SPLINE
SPL {X  -137.039, Y  +756.986, Z    +0.000, E1   -45.206, E3 +141112.390}
SPL {X  -152.094, Y  +724.074, Z    +0.000, E1   -34.132, E3 +141128.337}
SPL {X  -158.930, Y  +692.872, Z    +0.000, E1   -16.505, E3 +141134.653}
SPL {X  -160.000, Y  +673.072, Z    +0.000, E1    -0.858, E3 +141135.963}
SPL {X  -160.000, Y  +670.505, Z    +0.000, E1    +2.991, E3 +141136.000}
SPL {X  -160.000, Y  +665.157, Z    +0.000, E1   +13.199, E3 +141136.230}
SPL {X  -160.000, Y  +657.552, Z    +0.000, E1   +28.428, E3 +141136.915}
SPL {X  -160.000, Y  +642.088, Z    +0.000, E1   +49.428, E3 +141139.905}
SPL {X  -160.000, Y  +582.331, Z    +0.000, E1   +67.139, E3 +141162.371}
SPL {X  -160.000, Y  +443.344, Z    +0.000, E1   +69.515, E3 +141246.858}
SPL {X  -160.000, Y  +423.295, Z    +0.000, E1   +69.546, E3 +141262.678}
SPL {X  -155.937, Y  +349.874, Z    +0.000, E1   +73.941, E3 +141270.748}
SPL {X  -155.646, Y  +348.628, Z    +0.000, E1   +73.073, E3 +141280.631}
SPL {X  -155.163, Y  +346.655, Z    +0.000, E1   +71.976, E3 +141292.619}
SPL {X  -154.105, Y  +342.669, Z    +0.000, E1   +70.814, E3 +141306.124}
SPL {X  -152.951, Y  +338.733, Z    +0.000, E1   +69.529, E3 +141319.967}
SPL {X  -150.673, Y  +331.871, Z    +0.000, E1   +68.778, E3 +141331.215}
SPL {X  -146.876, Y  +322.238, Z    +0.000, E1   +68.294, E3 +141342.396}
SPL {X  -142.952, Y  +313.834, Z    +0.000, E1   +67.744, E3 +141352.675}
SPL {X  -139.245, Y  +306.891, Z    +0.000, E1   +67.208, E3 +141361.459}
SPL {X  -135.108, Y  +299.992, Z    +0.000, E1   +66.599, E3 +141370.410}
SPL {X  -130.642, Y  +293.328, Z    +0.000, E1   +65.888, E3 +141379.263}
SPL {X  -126.461, Y  +287.682, Z    +0.000, E1   +65.179, E3 +141386.826}
SPL {X   -93.259, Y  +255.690, Z    +0.000, E1   +54.095, E3 +141502.207}
ENDSPLINE

SPLINE
SPL {X  -130.811, Y  +293.568, Z    +0.000, E1   +46.951, E3 +141646.068}
SPL {X  -151.580, Y  +334.479, Z    +0.000, E1   +34.520, E3 +141670.191}
SPL {X  -157.897, Y  +359.846, Z    +0.000, E1   +21.040, E3 +141676.148}
SPL {X  -159.671, Y  +375.443, Z    +0.000, E1   +10.084, E3 +141677.964}
SPL {X  -160.000, Y  +387.403, Z    +0.000, E1    +0.377, E3 +141678.439}
SPL {X  -160.000, Y  +391.807, Z    +0.000, E1    -7.102, E3 +141678.543}
SPL {X  -160.000, Y  +398.244, Z    +0.000, E1   -19.803, E3 +141678.977}
SPL {X  -160.000, Y  +410.795, Z    +0.000, E1   -41.112, E3 +141680.790}
SPL {X  -160.000, Y  +461.796, Z    +0.000, E1   -65.564, E3 +141697.433}
SPL {X  -160.000, Y  +623.854, Z    +0.000, E1   -69.845, E3 +141791.505}
SPL {X  -160.000, Y  +641.581, Z    +0.000, E1   -69.837, E3 +141805.345}
SPL {X  -160.000, Y  +657.932, Z    +0.000, E1   -69.833, E3 +141818.103}
SPL {X  -159.989, Y  +676.310, Z    +0.000, E1   -69.844, E3 +141832.411}
SPL {X  -158.945, Y  +692.747, Z    +0.000, E1   -69.717, E3 +141846.339}
SPL {X  -156.998, Y  +705.248, Z    +0.000, E1   -69.481, E3 +141858.126}
SPL {X  -153.152, Y  +720.707, Z    +0.000, E1   -69.072, E3 +141874.038}
SPL {X  -148.823, Y  +733.152, Z    +0.000, E1   -68.450, E3 +141888.196}
SPL {X  -145.304, Y  +741.384, Z    +0.000, E1   -67.989, E3 +141897.996}
SPL {X  -141.481, Y  +749.119, Z    +0.000, E1   -67.448, E3 +141907.621}
SPL {X  -137.717, Y  +755.849, Z    +0.000, E1   -66.896, E3 +141916.255}
SPL {X  -133.615, Y  +762.417, Z    +0.000, E1   -66.275, E3 +141924.870}
SPL {X  -128.952, Y  +769.117, Z    +0.000, E1   -65.522, E3 +141933.832}
SPL {X  -125.615, Y  +773.501, Z    +0.000, E1   -64.909, E3 +141939.768}
SPL {X   -93.482, Y  +804.250, Z    +0.000, E1   -52.853, E3 +142076.966}
ENDSPLINE

SPLINE
SPL {X  -137.039, Y  +756.986, Z    +0.000, E1   -45.206, E3 +142207.629}
SPL {X  -152.094, Y  +724.074, Z    +0.000, E1   -34.132, E3 +142223.576}
SPL {X  -158.930, Y  +692.872, Z    +0.000, E1   -16.505, E3 +142229.892}
SPL {X  -160.000, Y  +673.072, Z    +0.000, E1    -0.858, E3 +142231.202}
SPL {X  -160.000, Y  +670.505, Z    +0.000, E1    +2.991, E3 +142231.239}
SPL {X  -160.000, Y  +665.157, Z    +0.000, E1   +13.199, E3 +142231.468}
SPL {X  -160.000, Y  +657.552, Z    +0.000, E1   +28.428, E3 +142232.153}
SPL {X  -160.000, Y  +642.088, Z    +0.000, E1   +49.428, E3 +142235.143}
SPL {X  -160.000, Y  +582.331, Z    +0.000, E1   +67.139, E3 +142257.610}
SPL {X  -160.000, Y  +443.344, Z    +0.000, E1   +69.515, E3 +142342.096}
SPL {X  -160.000, Y  +423.295, Z    +0.000, E1   +69.546, E3 +142357.917}
SPL {X  -155.937, Y  +349.874, Z    +0.000, E1   +73.941, E3 +142365.987}
SPL {X  -155.646, Y  +348.628, Z    +0.000, E1   +73.073, E3 +142375.870}
SPL {X  -155.163, Y  +346.655, Z    +0.000, E1   +71.976, E3 +142387.858}
SPL {X  -154.105, Y  +342.669, Z    +0.000, E1   +70.814, E3 +142401.363}
SPL {X  -152.951, Y  +338.733, Z    +0.000, E1   +69.529, E3 +142415.206}
SPL {X  -150.673, Y  +331.871, Z    +0.000, E1   +68.778, E3 +142426.454}
SPL {X  -146.876, Y  +322.238, Z    +0.000, E1   +68.294, E3 +142437.635}
SPL {X  -142.952, Y  +313.834, Z    +0.000, E1   +67.744, E3 +142447.914}
SPL {X  -139.245, Y  +306.891, Z    +0.000, E1   +67.208, E3 +142456.698}
SPL {X  -135.108, Y  +299.992, Z    +0.000, E1   +66.599, E3 +142465.649}
SPL {X  -130.642, Y  +293.328, Z    +0.000, E1   +65.888, E3 +142474.501}
SPL {X  -126.461, Y  +287.682, Z    +0.000, E1   +65.179, E3 +142482.064}
SPL {X   -93.259, Y  +255.690, Z    +0.000, E1   +54.095, E3 +142597.446}
ENDSPLINE

SPLINE
SPL {X  -130.811, Y  +293.568, Z    +0.000, E1   +46.951, E3 +142741.307}
SPL {X  -151.580, Y  +334.479, Z    +0.000, E1   +34.520, E3 +142765.429}
SPL {X  -157.897, Y  +359.846, Z    +0.000, E1   +21.040, E3 +142771.387}
SPL {X  -159.671, Y  +375.443, Z    +0.000, E1   +10.084, E3 +142773.202}
SPL {X  -160.000, Y  +387.403, Z    +0.000, E1    +0.377, E3 +142773.678}
SPL {X  -160.000, Y  +391.807, Z    +0.000, E1    -7.102, E3 +142773.782}
SPL {X  -160.000, Y  +398.244, Z    +0.000, E1   -19.803, E3 +142774.216}
SPL {X  -160.000, Y  +410.795, Z    +0.000, E1   -41.112, E3 +142776.029}
SPL {X  -160.000, Y  +461.796, Z    +0.000, E1   -65.564, E3 +142792.672}
SPL {X  -160.000, Y  +623.854, Z    +0.000, E1   -69.845, E3 +142886.744}
SPL {X  -160.000, Y  +641.581, Z    +0.000, E1   -69.837, E3 +142900.583}
SPL {X  -160.000, Y  +657.932, Z    +0.000, E1   -69.833, E3 +142913.342}
SPL {X  -159.989, Y  +676.310, Z    +0.000, E1   -69.844, E3 +142927.650}
SPL {X  -158.945, Y  +692.747, Z    +0.000, E1   -69.717, E3 +142941.578}
SPL {X  -156.998, Y  +705.248, Z    +0.000, E1   -69.481, E3 +142953.365}
SPL {X  -153.152, Y  +720.707, Z    +0.000, E1   -69.072, E3 +142969.276}
SPL {X  -148.823, Y  +733.152, Z    +0.000, E1   -68.450, E3 +142983.435}
SPL {X  -145.304, Y  +741.384, Z    +0.000, E1   -67.989, E3 +142993.235}
SPL {X  -141.481, Y  +749.119, Z    +0.000, E1   -67.448, E3 +143002.860}
SPL {X  -137.717, Y  +755.849, Z    +0.000, E1   -66.896, E3 +143011.494}
SPL {X  -133.615, Y  +762.417, Z    +0.000, E1   -66.275, E3 +143020.109}
SPL {X  -128.952, Y  +769.117, Z    +0.000, E1   -65.522, E3 +143029.070}
SPL {X  -125.615, Y  +773.501, Z    +0.000, E1   -64.909, E3 +143035.007}
SPL {X   -93.482, Y  +804.250, Z    +0.000, E1   -52.853, E3 +143172.205}
ENDSPLINE

SPLINE
SPL {X  -137.039, Y  +756.986, Z    +0.000, E1   -45.206, E3 +143302.868}
SPL {X  -152.094, Y  +724.074, Z    +0.000, E1   -34.132, E3 +143318.815}
SPL {X  -158.930, Y  +692.872, Z    +0.000, E1   -16.505, E3 +143325.130}
SPL {X  -160.000, Y  +673.072, Z    +0.000, E1    -0.858, E3 +143326.441}
SPL {X  -160.000, Y  +670.505, Z    +0.000, E1    +2.991, E3 +143326.477}
SPL {X  -160.000, Y  +665.157, Z    +0.000, E1   +13.199, E3 +143326.707}
SPL {X  -160.000, Y  +657.552, Z    +0.000, E1   +28.428, E3 +143327.392}
SPL {X  -160.000, Y  +642.088, Z    +0.000, E1   +49.428, E3 +143330.382}
SPL {X  -160.000, Y  +582.331, Z    +0.000, E1   +67.139, E3 +143352.849}
SPL {X  -160.000, Y  +443.344, Z    +0.000, E1   +69.515, E3 +143437.335}
SPL {X  -160.000, Y  +423.295, Z    +0.000, E1   +69.546, E3 +143453.155}
SPL {X  -155.937, Y  +349.874, Z    +0.000, E1   +73.941, E3 +143461.226}
SPL {X  -155.646, Y  +348.628, Z    +0.000, E1   +73.073, E3 +143471.109}
SPL {X  -155.163, Y  +346.655, Z    +0.000, E1   +71.976, E3 +143483.096}
SPL {X  -154.105, Y  +342.669, Z    +0.000, E1   +70.814, E3 +143496.601}
SPL {X  -152.951, Y  +338.733, Z    +0.000, E1   +69.529, E3 +143510.445}
SPL {X  -150.673, Y  +331.871, Z    +0.000, E1   +68.778, E3 +143521.693}
SPL {X  -146.876, Y  +322.238, Z    +0.000, E1   +68.294, E3 +143532.874}
SPL {X  -142.952, Y  +313.834, Z    +0.000, E1   +67.744, E3 +143543.153}
SPL {X  -139.245, Y  +306.891, Z    +0.000, E1   +67.208, E3 +143551.936}
SPL {X  -135.108, Y  +299.992, Z    +0.000, E1   +66.599, E3 +143560.888}
SPL {X  -130.642, Y  +293.328, Z    +0.000, E1   +65.888, E3 +143569.740}
SPL {X  -126.461, Y  +287.682, Z    +0.000, E1   +65.179, E3 +143577.303}
SPL {X   -93.259, Y  +255.690, Z    +0.000, E1   +54.095, E3 +143692.685}
ENDSPLINE

SPLINE
SPL {X  -130.811, Y  +293.568, Z    +0.000, E1   +46.951, E3 +143836.545}
SPL {X  -151.580, Y  +334.479, Z    +0.000, E1   +34.520, E3 +143860.668}
SPL {X  -157.897, Y  +359.846, Z    +0.000, E1   +21.040, E3 +143866.626}
SPL {X  -159.671, Y  +375.443, Z    +0.000, E1   +10.084, E3 +143868.441}
SPL {X  -160.000, Y  +387.403, Z    +0.000, E1    +0.377, E3 +143868.916}
SPL {X  -160.000, Y  +391.807, Z    +0.000, E1    -7.102, E3 +143869.021}
SPL {X  -160.000, Y  +398.244, Z    +0.000, E1   -19.803, E3 +143869.455}
SPL {X  -160.000, Y  +410.795, Z    +0.000, E1   -41.112, E3 +143871.267}
SPL {X  -160.000, Y  +461.796, Z    +0.000, E1   -65.564, E3 +143887.910}
SPL {X  -160.000, Y  +623.854, Z    +0.000, E1   -69.845, E3 +143981.983}
SPL {X  -160.000, Y  +641.581, Z    +0.000, E1   -69.837, E3 +143995.822}
SPL {X  -160.000, Y  +657.932, Z    +0.000, E1   -69.833, E3 +144008.580}
SPL {X  -159.989, Y  +676.310, Z    +0.000, E1   -69.844, E3 +144022.889}
SPL {X  -158.945, Y  +692.747, Z    +0.000, E1   -69.717, E3 +144036.816}
SPL {X  -156.998, Y  +705.248, Z    +0.000, E1   -69.481, E3 +144048.603}
SPL {X  -153.152, Y  +720.707, Z    +0.000, E1   -69.072, E3 +144064.515}
SPL {X  -148.823, Y  +733.152, Z    +0.000, E1   -68.450, E3 +144078.674}
SPL {X  -145.304, Y  +741.384, Z    +0.000, E1   -67.989, E3 +144088.474}
SPL {X  -141.481, Y  +749.119, Z    +0.000, E1   -67.448, E3 +144098.098}
SPL {X  -137.717, Y  +755.849, Z    +0.000, E1   -66.896, E3 +144106.733}
SPL {X  -133.615, Y  +762.417, Z    +0.000, E1   -66.275, E3 +144115.347}
SPL {X  -128.952, Y  +769.117, Z    +0.000, E1   -65.522, E3 +144124.309}
SPL {X  -125.615, Y  +773.501, Z    +0.000, E1   -64.909, E3 +144130.246}
SPL {X   -93.482, Y  +804.250, Z    +0.000, E1   -52.853, E3 +144267.443}
ENDSPLINE

SPLINE
SPL {X  -137.039, Y  +756.986, Z    +0.000, E1   -45.206, E3 +144398.106}
SPL {X  -152.094, Y  +724.074, Z    +0.000, E1   -34.132, E3 +144414.053}
SPL {X  -158.930, Y  +692.872, Z    +0.000, E1   -16.505, E3 +144420.369}
SPL {X  -160.000, Y  +673.072, Z    +0.000, E1    -0.858, E3 +144421.679}
SPL {X  -160.000, Y  +670.505, Z    +0.000, E1    +2.991, E3 +144421.716}
SPL {X  -160.000, Y  +665.157, Z    +0.000, E1   +13.199, E3 +144421.946}
SPL {X  -160.000, Y  +657.552, Z    +0.000, E1   +28.428, E3 +144422.631}
SPL {X  -160.000, Y  +642.088, Z    +0.000, E1   +49.428, E3 +144425.621}
SPL {X  -160.000, Y  +582.331, Z    +0.000, E1   +67.139, E3 +144448.087}
SPL {X  -160.000, Y  +443.344, Z    +0.000, E1   +69.515, E3 +144532.574}
SPL {X  -160.000, Y  +423.295, Z    +0.000, E1   +69.546, E3 +144548.394}
SPL {X  -155.937, Y  +349.874, Z    +0.000, E1   +73.941, E3 +144556.464}
SPL {X  -155.646, Y  +348.628, Z    +0.000, E1   +73.073, E3 +144566.347}
SPL {X  -155.163, Y  +346.655, Z    +0.000, E1   +71.976, E3 +144578.335}
SPL {X  -154.105, Y  +342.669, Z    +0.000, E1   +70.814, E3 +144591.840}
SPL {X  -152.951, Y  +338.733, Z    +0.000, E1   +69.529, E3 +144605.683}
ENDSPLINE

SPLINE
SPL {X  -155.937, Y  +349.872, Z    +0.000, E1   +65.931, E3 +143624.970}
SPL {X  -152.875, Y  +338.486, Z    +0.000, E1   +65.488, E3 +143638.669}
SPL {X  -149.360, Y  +328.327, Z    +0.000, E1   +64.994, E3 +143651.576}
SPL {X  -145.195, Y  +318.481, Z    +0.000, E1   +64.365, E3 +143664.729}
SPL {X  -140.564, Y  +309.268, Z    +0.000, E1   +63.646, E3 +143677.550}
SPL {X  -135.770, Y  +301.044, Z    +0.000, E1   +62.840, E3 +143689.422}
SPL {X  -130.944, Y  +293.756, Z    +0.000, E1   +61.990, E3 +143700.165}
SPL {X  -103.957, Y  +264.074, Z    +0.000, E1   +52.557, E3 +143806.269}
ENDSPLINE

SPLINE
SPL {X  -133.093, Y  +296.896, Z    +0.000, E1   +44.059, E3 +143931.102}
SPL {X  -150.601, Y  +331.670, Z    +0.000, E1   +33.435, E3 +143955.365}
SPL {X  -157.739, Y  +358.898, Z    +0.000, E1   +20.026, E3 +143963.593}
SPL {X  -159.601, Y  +374.403, Z    +0.000, E1   +10.058, E3 +143965.908}
SPL {X  -159.993, Y  +384.251, Z    +0.000, E1    +2.830, E3 +143966.540}
SPL {X  -160.000, Y  +387.929, Z    +0.000, E1    -0.363, E3 +143966.609}
SPL {X  -160.000, Y  +392.137, Z    +0.000, E1    -6.580, E3 +143966.748}
SPL {X  -160.000, Y  +398.334, Z    +0.000, E1   -17.404, E3 +143967.239}
SPL {X  -160.000, Y  +410.558, Z    +0.000, E1   -36.649, E3 +143969.342}
SPL {X  -160.000, Y  +459.534, Z    +0.000, E1   -61.429, E3 +143988.937}
SPL {X  -160.000, Y  +586.246, Z    +0.000, E1   -66.315, E3 +144075.436}
SPL {X  -160.000, Y  +602.823, Z    +0.000, E1   -66.332, E3 +144090.840}
SPL {X  -160.000, Y  +621.796, Z    +0.000, E1   -66.332, E3 +144108.509}
SPL {X  -160.000, Y  +638.226, Z    +0.000, E1   -66.314, E3 +144123.837}
SPL {X  -160.000, Y  +655.092, Z    +0.000, E1   -66.336, E3 +144139.495}
SPL {X  -160.000, Y  +671.716, Z    +0.000, E1   -66.315, E3 +144155.009}
SPL {X  -159.502, Y  +687.017, Z    +0.000, E1   -66.266, E3 +144169.759}
SPL {X  -157.713, Y  +701.353, Z    +0.000, E1   -66.026, E3 +144184.986}
SPL {X  -155.081, Y  +713.767, Z    +0.000, E1   -65.665, E3 +144199.272}
SPL {X  -152.128, Y  +723.968, Z    +0.000, E1   -65.242, E3 +144211.771}
SPL {X  -148.925, Y  +732.892, Z    +0.000, E1   -64.779, E3 +144223.271}
SPL {X  -144.887, Y  +742.280, Z    +0.000, E1   -64.184, E3 +144235.901}
SPL {X  -140.317, Y  +751.285, Z    +0.000, E1   -63.454, E3 +144248.538}
SPL {X  -135.706, Y  +759.158, Z    +0.000, E1   -62.682, E3 +144259.939}
SPL {X  -131.040, Y  +766.207, Z    +0.000, E1   -61.854, E3 +144270.371}
SPL {X  -102.962, Y  +796.870, Z    +0.000, E1   -51.620, E3 +144395.703}
ENDSPLINE

SPLINE
SPL {X  -139.855, Y  +752.122, Z    +0.000, E1   -42.075, E3 +144518.631}
SPL {X  -153.268, Y  +720.324, Z    +0.000, E1   -30.648, E3 +144534.877}
SPL {X  -158.910, Y  +693.048, Z    +0.000, E1   -15.531, E3 +144540.948}
SPL {X  -159.977, Y  +677.095, Z    +0.000, E1    -3.968, E3 +144542.371}
SPL {X  -160.000, Y  +672.556, Z    +0.000, E1    -0.073, E3 +144542.473}
SPL {X  -160.000, Y  +669.399, Z    +0.000, E1    +3.976, E3 +144542.553}
SPL {X  -160.000, Y  +661.045, Z    +0.000, E1   +19.300, E3 +144543.142}
SPL {X  -160.000, Y  +646.999, Z    +0.000, E1   +41.048, E3 +144545.559}
SPL {X  -160.000, Y  +594.464, Z    +0.000, E1   +63.651, E3 +144565.860}
SPL {X  -160.000, Y  +465.200, Z    +0.000, E1   +67.027, E3 +144654.430}
SPL {X  -160.000, Y  +444.745, Z    +0.000, E1   +67.032, E3 +144672.838}
SPL {X  -160.000, Y  +422.224, Z    +0.000, E1   +67.044, E3 +144693.090}
ENDSPLINE

SPLINE
SPL {X  -160.000, Y  +424.635, Z    +0.000, E1   +64.425, E3 +144711.117}
ENDSPLINE

SPLINE
SPL {X  -160.000, Y  +410.501, Z    +0.000, E1   +64.162, E3 +144727.661}
SPL {X  -160.000, Y  +387.965, Z    +0.000, E1   +65.039, E3 +144743.613}
SPL {X  -158.836, Y  +366.435, Z    +0.000, E1   +65.805, E3 +144758.554}
SPL {X  -155.922, Y  +349.806, Z    +0.000, E1   +65.927, E3 +144773.200}
SPL {X  -152.875, Y  +338.486, Z    +0.000, E1   +65.488, E3 +144786.817}
SPL {X  -149.360, Y  +328.327, Z    +0.000, E1   +64.994, E3 +144799.724}
SPL {X  -145.195, Y  +318.481, Z    +0.000, E1   +64.365, E3 +144812.877}
SPL {X  -140.564, Y  +309.268, Z    +0.000, E1   +63.646, E3 +144825.698}
SPL {X  -135.770, Y  +301.044, Z    +0.000, E1   +62.840, E3 +144837.569}
SPL {X  -130.944, Y  +293.756, Z    +0.000, E1   +61.990, E3 +144848.313}
SPL {X  -103.957, Y  +264.074, Z    +0.000, E1   +52.557, E3 +144954.416}
ENDSPLINE

SPLINE
SPL {X  -133.093, Y  +296.896, Z    +0.000, E1   +44.059, E3 +145079.250}
SPL {X  -150.601, Y  +331.670, Z    +0.000, E1   +33.435, E3 +145103.513}
SPL {X  -157.739, Y  +358.898, Z    +0.000, E1   +20.026, E3 +145111.741}
SPL {X  -159.601, Y  +374.403, Z    +0.000, E1   +10.058, E3 +145114.056}
SPL {X  -159.993, Y  +384.251, Z    +0.000, E1    +2.830, E3 +145114.688}
SPL {X  -160.000, Y  +387.929, Z    +0.000, E1    -0.363, E3 +145114.757}
SPL {X  -160.000, Y  +392.137, Z    +0.000, E1    -6.580, E3 +145114.895}
SPL {X  -160.000, Y  +398.334, Z    +0.000, E1   -17.404, E3 +145115.387}
SPL {X  -160.000, Y  +410.558, Z    +0.000, E1   -36.649, E3 +145117.490}
SPL {X  -160.000, Y  +459.534, Z    +0.000, E1   -61.429, E3 +145137.085}
SPL {X  -160.000, Y  +586.246, Z    +0.000, E1   -66.315, E3 +145223.584}
SPL {X  -160.000, Y  +602.823, Z    +0.000, E1   -66.332, E3 +145238.988}
SPL {X  -160.000, Y  +621.796, Z    +0.000, E1   -66.332, E3 +145256.657}
SPL {X  -160.000, Y  +638.226, Z    +0.000, E1   -66.314, E3 +145271.984}
SPL {X  -160.000, Y  +655.092, Z    +0.000, E1   -66.336, E3 +145287.643}
SPL {X  -160.000, Y  +671.716, Z    +0.000, E1   -66.315, E3 +145303.157}
SPL {X  -159.502, Y  +687.017, Z    +0.000, E1   -66.266, E3 +145317.907}
SPL {X  -157.713, Y  +701.353, Z    +0.000, E1   -66.026, E3 +145333.134}
SPL {X  -155.081, Y  +713.767, Z    +0.000, E1   -65.665, E3 +145347.420}
SPL {X  -152.128, Y  +723.968, Z    +0.000, E1   -65.242, E3 +145359.919}
SPL {X  -148.925, Y  +732.892, Z    +0.000, E1   -64.779, E3 +145371.419}
SPL {X  -144.887, Y  +742.280, Z    +0.000, E1   -64.184, E3 +145384.049}
SPL {X  -140.317, Y  +751.285, Z    +0.000, E1   -63.454, E3 +145396.686}
SPL {X  -135.706, Y  +759.158, Z    +0.000, E1   -62.682, E3 +145408.087}
SPL {X  -131.040, Y  +766.207, Z    +0.000, E1   -61.854, E3 +145418.519}
SPL {X  -102.962, Y  +796.870, Z    +0.000, E1   -51.620, E3 +145543.851}
ENDSPLINE

SPLINE
SPL {X  -139.855, Y  +752.122, Z    +0.000, E1   -42.075, E3 +145666.779}
SPL {X  -153.268, Y  +720.324, Z    +0.000, E1   -30.648, E3 +145683.025}
SPL {X  -158.910, Y  +693.048, Z    +0.000, E1   -15.531, E3 +145689.096}
SPL {X  -159.977, Y  +677.095, Z    +0.000, E1    -3.968, E3 +145690.519}
SPL {X  -160.000, Y  +672.556, Z    +0.000, E1    -0.073, E3 +145690.621}
SPL {X  -160.000, Y  +669.399, Z    +0.000, E1    +3.976, E3 +145690.701}
SPL {X  -160.000, Y  +661.045, Z    +0.000, E1   +19.300, E3 +145691.290}
SPL {X  -160.000, Y  +646.999, Z    +0.000, E1   +41.048, E3 +145693.707}
SPL {X  -160.000, Y  +594.464, Z    +0.000, E1   +63.651, E3 +145714.007}
SPL {X  -160.000, Y  +465.200, Z    +0.000, E1   +67.027, E3 +145802.578}
SPL {X  -160.000, Y  +444.745, Z    +0.000, E1   +67.032, E3 +145820.986}
SPL {X  -160.000, Y  +422.224, Z    +0.000, E1   +67.044, E3 +145841.238}
ENDSPLINE

SPLINE
SPL {X  -160.000, Y  +424.635, Z    +0.000, E1   +64.425, E3 +145859.265}
ENDSPLINE

SPLINE
SPL {X  -160.000, Y  +410.501, Z    +0.000, E1   +64.162, E3 +145875.809}
SPL {X  -160.000, Y  +387.965, Z    +0.000, E1   +65.039, E3 +145891.761}
SPL {X  -158.836, Y  +366.435, Z    +0.000, E1   +65.805, E3 +145906.702}
SPL {X  -155.922, Y  +349.806, Z    +0.000, E1   +65.927, E3 +145921.348}
SPL {X  -152.875, Y  +338.486, Z    +0.000, E1   +65.488, E3 +145934.965}
SPL {X  -149.360, Y  +328.327, Z    +0.000, E1   +64.994, E3 +145947.872}
SPL {X  -145.195, Y  +318.481, Z    +0.000, E1   +64.365, E3 +145961.025}
SPL {X  -140.564, Y  +309.268, Z    +0.000, E1   +63.646, E3 +145973.846}
SPL {X  -135.770, Y  +301.044, Z    +0.000, E1   +62.840, E3 +145985.717}
SPL {X  -130.944, Y  +293.756, Z    +0.000, E1   +61.990, E3 +145996.460}
SPL {X  -103.957, Y  +264.074, Z    +0.000, E1   +52.557, E3 +146102.564}
ENDSPLINE

SPLINE
SPL {X  -133.093, Y  +296.896, Z    +0.000, E1   +44.059, E3 +146227.398}
SPL {X  -150.601, Y  +331.670, Z    +0.000, E1   +33.435, E3 +146251.661}
SPL {X  -157.739, Y  +358.898, Z    +0.000, E1   +20.026, E3 +146259.889}
SPL {X  -159.601, Y  +374.403, Z    +0.000, E1   +10.058, E3 +146262.204}
SPL {X  -159.993, Y  +384.251, Z    +0.000, E1    +2.830, E3 +146262.836}
SPL {X  -160.000, Y  +387.929, Z    +0.000, E1    -0.363, E3 +146262.905}
SPL {X  -160.000, Y  +392.137, Z    +0.000, E1    -6.580, E3 +146263.043}
SPL {X  -160.000, Y  +398.334, Z    +0.000, E1   -17.404, E3 +146263.535}
SPL {X  -160.000, Y  +410.558, Z    +0.000, E1   -36.649, E3 +146265.638}
SPL {X  -160.000, Y  +459.534, Z    +0.000, E1   -61.429, E3 +146285.233}
SPL {X  -160.000, Y  +586.246, Z    +0.000, E1   -66.315, E3 +146371.732}
SPL {X  -160.000, Y  +602.823, Z    +0.000, E1   -66.332, E3 +146387.136}
SPL {X  -160.000, Y  +621.796, Z    +0.000, E1   -66.332, E3 +146404.805}
SPL {X  -160.000, Y  +638.226, Z    +0.000, E1   -66.314, E3 +146420.132}
SPL {X  -160.000, Y  +655.092, Z    +0.000, E1   -66.336, E3 +146435.791}
SPL {X  -160.000, Y  +671.716, Z    +0.000, E1   -66.315, E3 +146451.305}
SPL {X  -159.502, Y  +687.017, Z    +0.000, E1   -66.266, E3 +146466.055}
SPL {X  -157.713, Y  +701.353, Z    +0.000, E1   -66.026, E3 +146481.282}
SPL {X  -155.081, Y  +713.767, Z    +0.000, E1   -65.665, E3 +146495.568}
SPL {X  -152.128, Y  +723.968, Z    +0.000, E1   -65.242, E3 +146508.067}
SPL {X  -148.925, Y  +732.892, Z    +0.000, E1   -64.779, E3 +146519.567}
SPL {X  -144.887, Y  +742.280, Z    +0.000, E1   -64.184, E3 +146532.197}
SPL {X  -140.317, Y  +751.285, Z    +0.000, E1   -63.454, E3 +146544.834}
SPL {X  -135.706, Y  +759.158, Z    +0.000, E1   -62.682, E3 +146556.235}
SPL {X  -131.040, Y  +766.207, Z    +0.000, E1   -61.854, E3 +146566.667}
SPL {X  -102.962, Y  +796.870, Z    +0.000, E1   -51.620, E3 +146691.999}
ENDSPLINE

SPLINE
SPL {X  -139.855, Y  +752.122, Z    +0.000, E1   -42.075, E3 +146814.927}
SPL {X  -153.268, Y  +720.324, Z    +0.000, E1   -30.648, E3 +146831.173}
SPL {X  -158.910, Y  +693.048, Z    +0.000, E1   -15.531, E3 +146837.243}
SPL {X  -159.977, Y  +677.095, Z    +0.000, E1    -3.968, E3 +146838.667}
SPL {X  -160.000, Y  +672.556, Z    +0.000, E1    -0.073, E3 +146838.769}
SPL {X  -160.000, Y  +669.399, Z    +0.000, E1    +3.976, E3 +146838.849}
SPL {X  -160.000, Y  +661.045, Z    +0.000, E1   +19.300, E3 +146839.438}
SPL {X  -160.000, Y  +646.999, Z    +0.000, E1   +41.048, E3 +146841.855}
SPL {X  -160.000, Y  +594.464, Z    +0.000, E1   +63.651, E3 +146862.155}
SPL {X  -160.000, Y  +465.200, Z    +0.000, E1   +67.027, E3 +146950.726}
SPL {X  -160.000, Y  +444.745, Z    +0.000, E1   +67.032, E3 +146969.134}
SPL {X  -160.000, Y  +422.224, Z    +0.000, E1   +67.044, E3 +146989.386}
ENDSPLINE

SPLINE
SPL {X  -160.000, Y  +424.635, Z    +0.000, E1   +64.425, E3 +147007.413}
ENDSPLINE

SPLINE
SPL {X  -160.000, Y  +410.501, Z    +0.000, E1   +64.162, E3 +147023.957}
SPL {X  -160.000, Y  +387.965, Z    +0.000, E1   +65.039, E3 +147039.909}
SPL {X  -158.836, Y  +366.435, Z    +0.000, E1   +65.805, E3 +147054.850}
SPL {X  -155.922, Y  +349.806, Z    +0.000, E1   +65.927, E3 +147069.496}
SPL {X  -152.875, Y  +338.486, Z    +0.000, E1   +65.488, E3 +147083.113}
SPL {X  -149.360, Y  +328.327, Z    +0.000, E1   +64.994, E3 +147096.019}
SPL {X  -145.195, Y  +318.481, Z    +0.000, E1   +64.365, E3 +147109.173}
SPL {X  -140.564, Y  +309.268, Z    +0.000, E1   +63.646, E3 +147121.994}
SPL {X  -135.770, Y  +301.044, Z    +0.000, E1   +62.840, E3 +147133.865}
SPL {X  -130.944, Y  +293.756, Z    +0.000, E1   +61.990, E3 +147144.608}
SPL {X  -103.957, Y  +264.074, Z    +0.000, E1   +52.557, E3 +147250.712}
ENDSPLINE

SPLINE
SPL {X  -133.093, Y  +296.896, Z    +0.000, E1   +44.059, E3 +147375.546}
SPL {X  -150.601, Y  +331.670, Z    +0.000, E1   +33.435, E3 +147399.809}
SPL {X  -157.739, Y  +358.898, Z    +0.000, E1   +20.026, E3 +147408.037}
SPL {X  -159.601, Y  +374.403, Z    +0.000, E1   +10.058, E3 +147410.352}
SPL {X  -159.993, Y  +384.251, Z    +0.000, E1    +2.830, E3 +147410.984}
SPL {X  -160.000, Y  +387.929, Z    +0.000, E1    -0.363, E3 +147411.053}
SPL {X  -160.000, Y  +392.137, Z    +0.000, E1    -6.580, E3 +147411.191}
SPL {X  -160.000, Y  +398.334, Z    +0.000, E1   -17.404, E3 +147411.683}
SPL {X  -160.000, Y  +410.558, Z    +0.000, E1   -36.649, E3 +147413.786}
SPL {X  -160.000, Y  +459.534, Z    +0.000, E1   -61.429, E3 +147433.381}
SPL {X  -160.000, Y  +586.246, Z    +0.000, E1   -66.315, E3 +147519.880}
SPL {X  -160.000, Y  +602.823, Z    +0.000, E1   -66.332, E3 +147535.284}
SPL {X  -160.000, Y  +621.796, Z    +0.000, E1   -66.332, E3 +147552.953}
SPL {X  -160.000, Y  +638.226, Z    +0.000, E1   -66.314, E3 +147568.280}
SPL {X  -160.000, Y  +655.092, Z    +0.000, E1   -66.336, E3 +147583.939}
SPL {X  -160.000, Y  +671.716, Z    +0.000, E1   -66.315, E3 +147599.453}
SPL {X  -159.502, Y  +687.017, Z    +0.000, E1   -66.266, E3 +147614.203}
SPL {X  -157.713, Y  +701.353, Z    +0.000, E1   -66.026, E3 +147629.430}
SPL {X  -155.081, Y  +713.767, Z    +0.000, E1   -65.665, E3 +147643.715}
SPL {X  -152.128, Y  +723.968, Z    +0.000, E1   -65.242, E3 +147656.215}
SPL {X  -148.925, Y  +732.892, Z    +0.000, E1   -64.779, E3 +147667.715}
SPL {X  -144.887, Y  +742.280, Z    +0.000, E1   -64.184, E3 +147680.345}
SPL {X  -140.317, Y  +751.285, Z    +0.000, E1   -63.454, E3 +147692.982}
SPL {X  -135.706, Y  +759.158, Z    +0.000, E1   -62.682, E3 +147704.383}
SPL {X  -131.040, Y  +766.207, Z    +0.000, E1   -61.854, E3 +147714.815}
SPL {X  -102.962, Y  +796.870, Z    +0.000, E1   -51.620, E3 +147840.147}
ENDSPLINE

SPLINE
SPL {X  -139.855, Y  +752.122, Z    +0.000, E1   -42.075, E3 +147963.075}
SPL {X  -153.268, Y  +720.324, Z    +0.000, E1   -30.648, E3 +147979.321}
SPL {X  -158.910, Y  +693.048, Z    +0.000, E1   -15.531, E3 +147985.391}
SPL {X  -159.977, Y  +677.095, Z    +0.000, E1    -3.968, E3 +147986.815}
SPL {X  -160.000, Y  +672.556, Z    +0.000, E1    -0.073, E3 +147986.917}
SPL {X  -160.000, Y  +669.399, Z    +0.000, E1    +3.976, E3 +147986.997}
SPL {X  -160.000, Y  +661.045, Z    +0.000, E1   +19.300, E3 +147987.586}
SPL {X  -160.000, Y  +646.999, Z    +0.000, E1   +41.048, E3 +147990.003}
SPL {X  -160.000, Y  +594.464, Z    +0.000, E1   +63.651, E3 +148010.303}
SPL {X  -160.000, Y  +465.200, Z    +0.000, E1   +67.027, E3 +148098.873}
SPL {X  -160.000, Y  +444.745, Z    +0.000, E1   +67.032, E3 +148117.282}
SPL {X  -160.000, Y  +422.224, Z    +0.000, E1   +67.044, E3 +148137.534}
ENDSPLINE

SPLINE
SPL {X  -160.000, Y  +424.635, Z    +0.000, E1   +64.425, E3 +148155.560}
ENDSPLINE

SPLINE
SPL {X  -160.000, Y  +410.501, Z    +0.000, E1   +64.162, E3 +148172.105}
SPL {X  -160.000, Y  +387.965, Z    +0.000, E1   +65.039, E3 +148188.057}
SPL {X  -158.836, Y  +366.435, Z    +0.000, E1   +65.805, E3 +148202.998}
SPL {X  -155.922, Y  +349.806, Z    +0.000, E1   +65.927, E3 +148217.644}
SPL {X  -152.875, Y  +338.486, Z    +0.000, E1   +65.488, E3 +148231.261}
SPL {X  -149.360, Y  +328.327, Z    +0.000, E1   +64.994, E3 +148244.167}
SPL {X  -145.195, Y  +318.481, Z    +0.000, E1   +64.365, E3 +148257.321}
SPL {X  -140.564, Y  +309.268, Z    +0.000, E1   +63.646, E3 +148270.142}
SPL {X  -135.770, Y  +301.044, Z    +0.000, E1   +62.840, E3 +148282.013}
SPL {X  -130.944, Y  +293.756, Z    +0.000, E1   +61.990, E3 +148292.756}
SPL {X  -103.957, Y  +264.074, Z    +0.000, E1   +52.557, E3 +148398.860}
ENDSPLINE

SPLINE
SPL {X  -133.093, Y  +296.896, Z    +0.000, E1   +44.059, E3 +148523.694}
SPL {X  -150.601, Y  +331.670, Z    +0.000, E1   +33.435, E3 +148547.957}
SPL {X  -157.739, Y  +358.898, Z    +0.000, E1   +20.026, E3 +148556.184}
SPL {X  -159.601, Y  +374.403, Z    +0.000, E1   +10.058, E3 +148558.500}
SPL {X  -159.993, Y  +384.251, Z    +0.000, E1    +2.830, E3 +148559.132}
SPL {X  -160.000, Y  +387.929, Z    +0.000, E1    -0.363, E3 +148559.200}
SPL {X  -160.000, Y  +392.137, Z    +0.000, E1    -6.580, E3 +148559.339}
SPL {X  -160.000, Y  +398.334, Z    +0.000, E1   -17.404, E3 +148559.831}
SPL {X  -160.000, Y  +410.558, Z    +0.000, E1   -36.649, E3 +148561.934}
SPL {X  -160.000, Y  +459.534, Z    +0.000, E1   -61.429, E3 +148581.528}
SPL {X  -160.000, Y  +586.246, Z    +0.000, E1   -66.315, E3 +148668.028}
SPL {X  -160.000, Y  +602.823, Z    +0.000, E1   -66.332, E3 +148683.432}
SPL {X  -160.000, Y  +621.796, Z    +0.000, E1   -66.332, E3 +148701.101}
SPL {X  -160.000, Y  +638.226, Z    +0.000, E1   -66.314, E3 +148716.428}
SPL {X  -160.000, Y  +655.092, Z    +0.000, E1   -66.336, E3 +148732.087}
SPL {X  -160.000, Y  +671.716, Z    +0.000, E1   -66.315, E3 +148747.601}
SPL {X  -159.502, Y  +687.017, Z    +0.000, E1   -66.266, E3 +148762.351}
SPL {X  -157.713, Y  +701.353, Z    +0.000, E1   -66.026, E3 +148777.578}
SPL {X  -155.081, Y  +713.767, Z    +0.000, E1   -65.665, E3 +148791.863}
SPL {X  -152.128, Y  +723.968, Z    +0.000, E1   -65.242, E3 +148804.363}
SPL {X  -148.925, Y  +732.892, Z    +0.000, E1   -64.779, E3 +148815.863}
SPL {X  -144.887, Y  +742.280, Z    +0.000, E1   -64.184, E3 +148828.492}
SPL {X  -140.317, Y  +751.285, Z    +0.000, E1   -63.454, E3 +148841.130}
SPL {X  -135.706, Y  +759.158, Z    +0.000, E1   -62.682, E3 +148852.531}
SPL {X  -131.040, Y  +766.207, Z    +0.000, E1   -61.854, E3 +148862.963}
SPL {X  -102.962, Y  +796.870, Z    +0.000, E1   -51.620, E3 +148988.295}
ENDSPLINE

SPLINE
SPL {X  -139.855, Y  +752.122, Z    +0.000, E1   -42.075, E3 +149111.223}
SPL {X  -153.268, Y  +720.324, Z    +0.000, E1   -30.648, E3 +149127.469}
SPL {X  -158.910, Y  +693.048, Z    +0.000, E1   -15.531, E3 +149133.539}
SPL {X  -159.977, Y  +677.095, Z    +0.000, E1    -3.968, E3 +149134.963}
SPL {X  -160.000, Y  +672.556, Z    +0.000, E1    -0.073, E3 +149135.065}
SPL {X  -160.000, Y  +669.399, Z    +0.000, E1    +3.976, E3 +149135.145}
SPL {X  -160.000, Y  +661.045, Z    +0.000, E1   +19.300, E3 +149135.733}
SPL {X  -160.000, Y  +646.999, Z    +0.000, E1   +41.048, E3 +149138.151}
SPL {X  -160.000, Y  +594.464, Z    +0.000, E1   +63.651, E3 +149158.451}
SPL {X  -160.000, Y  +465.200, Z    +0.000, E1   +67.027, E3 +149247.021}
SPL {X  -160.000, Y  +444.745, Z    +0.000, E1   +67.032, E3 +149265.430}
SPL {X  -160.000, Y  +422.224, Z    +0.000, E1   +67.044, E3 +149285.682}
ENDSPLINE

SPLINE
SPL {X  -160.000, Y  +424.635, Z    +0.000, E1   +64.425, E3 +149303.708}
ENDSPLINE

SPLINE
SPL {X  -160.000, Y  +410.501, Z    +0.000, E1   +64.162, E3 +149320.253}
SPL {X  -160.000, Y  +387.965, Z    +0.000, E1   +65.039, E3 +149336.205}
SPL {X  -158.836, Y  +366.435, Z    +0.000, E1   +65.805, E3 +149351.146}
SPL {X  -155.922, Y  +349.806, Z    +0.000, E1   +65.927, E3 +149365.792}
SPL {X  -152.875, Y  +338.486, Z    +0.000, E1   +65.488, E3 +149379.409}
SPL {X  -149.360, Y  +328.327, Z    +0.000, E1   +64.994, E3 +149392.315}
SPL {X  -145.195, Y  +318.481, Z    +0.000, E1   +64.365, E3 +149405.469}
SPL {X  -140.564, Y  +309.268, Z    +0.000, E1   +63.646, E3 +149418.290}
SPL {X  -135.770, Y  +301.044, Z    +0.000, E1   +62.840, E3 +149430.161}
SPL {X  -130.944, Y  +293.756, Z    +0.000, E1   +61.990, E3 +149440.904}
SPL {X  -103.957, Y  +264.074, Z    +0.000, E1   +52.557, E3 +149547.008}
ENDSPLINE

SPLINE
SPL {X  -133.093, Y  +296.896, Z    +0.000, E1   +44.059, E3 +149671.842}
SPL {X  -150.601, Y  +331.670, Z    +0.000, E1   +33.435, E3 +149696.105}
SPL {X  -157.739, Y  +358.898, Z    +0.000, E1   +20.026, E3 +149704.332}
SPL {X  -159.601, Y  +374.403, Z    +0.000, E1   +10.058, E3 +149706.648}
SPL {X  -159.993, Y  +384.251, Z    +0.000, E1    +2.830, E3 +149707.280}
SPL {X  -160.000, Y  +387.929, Z    +0.000, E1    -0.363, E3 +149707.348}
SPL {X  -160.000, Y  +392.137, Z    +0.000, E1    -6.580, E3 +149707.487}
SPL {X  -160.000, Y  +398.334, Z    +0.000, E1   -17.404, E3 +149707.979}
SPL {X  -160.000, Y  +410.558, Z    +0.000, E1   -36.649, E3 +149710.082}
SPL {X  -160.000, Y  +459.534, Z    +0.000, E1   -61.429, E3 +149729.676}
SPL {X  -160.000, Y  +586.246, Z    +0.000, E1   -66.315, E3 +149816.176}
SPL {X  -160.000, Y  +602.823, Z    +0.000, E1   -66.332, E3 +149831.580}
SPL {X  -160.000, Y  +621.796, Z    +0.000, E1   -66.332, E3 +149849.249}
SPL {X  -160.000, Y  +638.226, Z    +0.000, E1   -66.314, E3 +149864.576}
SPL {X  -160.000, Y  +655.092, Z    +0.000, E1   -66.336, E3 +149880.235}
SPL {X  -160.000, Y  +671.716, Z    +0.000, E1   -66.315, E3 +149895.749}
SPL {X  -159.502, Y  +687.017, Z    +0.000, E1   -66.266, E3 +149910.499}
SPL {X  -157.713, Y  +701.353, Z    +0.000, E1   -66.026, E3 +149925.726}
SPL {X  -155.081, Y  +713.767, Z    +0.000, E1   -65.665, E3 +149940.011}
SPL {X  -152.128, Y  +723.968, Z    +0.000, E1   -65.242, E3 +149952.511}
SPL {X  -148.925, Y  +732.892, Z    +0.000, E1   -64.779, E3 +149964.011}
SPL {X  -144.887, Y  +742.280, Z    +0.000, E1   -64.184, E3 +149976.640}
SPL {X  -140.317, Y  +751.285, Z    +0.000, E1   -63.454, E3 +149989.278}
SPL {X  -135.706, Y  +759.158, Z    +0.000, E1   -62.682, E3 +150000.679}
SPL {X  -131.040, Y  +766.207, Z    +0.000, E1   -61.854, E3 +150011.111}
SPL {X  -102.962, Y  +796.870, Z    +0.000, E1   -51.620, E3 +150136.443}
ENDSPLINE

SPLINE
SPL {X  -139.855, Y  +752.122, Z    +0.000, E1   -42.075, E3 +150259.371}
SPL {X  -153.268, Y  +720.324, Z    +0.000, E1   -30.648, E3 +150275.617}
SPL {X  -158.910, Y  +693.048, Z    +0.000, E1   -15.531, E3 +150281.687}
SPL {X  -159.977, Y  +677.095, Z    +0.000, E1    -3.968, E3 +150283.111}
SPL {X  -160.000, Y  +672.556, Z    +0.000, E1    -0.073, E3 +150283.213}
SPL {X  -160.000, Y  +669.399, Z    +0.000, E1    +3.976, E3 +150283.293}
SPL {X  -160.000, Y  +661.045, Z    +0.000, E1   +19.300, E3 +150283.881}
SPL {X  -160.000, Y  +646.999, Z    +0.000, E1   +41.048, E3 +150286.299}
SPL {X  -160.000, Y  +594.464, Z    +0.000, E1   +63.651, E3 +150306.599}
SPL {X  -160.000, Y  +465.200, Z    +0.000, E1   +67.027, E3 +150395.169}
SPL {X  -160.000, Y  +444.745, Z    +0.000, E1   +67.032, E3 +150413.578}
SPL {X  -160.000, Y  +422.224, Z    +0.000, E1   +67.044, E3 +150433.830}
ENDSPLINE

SPLINE
SPL {X  -160.000, Y  +424.635, Z    +0.000, E1   +64.425, E3 +150451.856}
ENDSPLINE

SPLINE
SPL {X  -160.000, Y  +410.501, Z    +0.000, E1   +64.162, E3 +150468.401}
SPL {X  -160.000, Y  +387.965, Z    +0.000, E1   +65.039, E3 +150484.352}
SPL {X  -158.836, Y  +366.435, Z    +0.000, E1   +65.805, E3 +150499.294}
SPL {X  -155.922, Y  +349.806, Z    +0.000, E1   +65.927, E3 +150513.940}
SPL {X  -152.875, Y  +338.486, Z    +0.000, E1   +65.488, E3 +150527.557}
SPL {X  -149.360, Y  +328.327, Z    +0.000, E1   +64.994, E3 +150540.463}
SPL {X  -145.195, Y  +318.481, Z    +0.000, E1   +64.365, E3 +150553.617}
SPL {X  -140.564, Y  +309.268, Z    +0.000, E1   +63.646, E3 +150566.438}
SPL {X  -135.770, Y  +301.044, Z    +0.000, E1   +62.840, E3 +150578.309}
SPL {X  -130.944, Y  +293.756, Z    +0.000, E1   +61.990, E3 +150589.052}
SPL {X  -103.957, Y  +264.074, Z    +0.000, E1   +52.557, E3 +150695.156}
ENDSPLINE

SPLINE
SPL {X  -133.093, Y  +296.896, Z    +0.000, E1   +44.059, E3 +150819.990}
SPL {X  -150.601, Y  +331.670, Z    +0.000, E1   +33.435, E3 +150844.252}
SPL {X  -157.739, Y  +358.898, Z    +0.000, E1   +20.026, E3 +150852.480}
SPL {X  -159.601, Y  +374.403, Z    +0.000, E1   +10.058, E3 +150854.796}
SPL {X  -159.993, Y  +384.251, Z    +0.000, E1    +2.830, E3 +150855.428}
SPL {X  -160.000, Y  +387.929, Z    +0.000, E1    -0.363, E3 +150855.496}
SPL {X  -160.000, Y  +392.137, Z    +0.000, E1    -6.580, E3 +150855.635}
SPL {X  -160.000, Y  +398.334, Z    +0.000, E1   -17.404, E3 +150856.127}
SPL {X  -160.000, Y  +410.558, Z    +0.000, E1   -36.649, E3 +150858.230}
SPL {X  -160.000, Y  +459.534, Z    +0.000, E1   -61.429, E3 +150877.824}
SPL {X  -160.000, Y  +586.246, Z    +0.000, E1   -66.315, E3 +150964.324}
SPL {X  -160.000, Y  +602.823, Z    +0.000, E1   -66.332, E3 +150979.728}
SPL {X  -160.000, Y  +621.796, Z    +0.000, E1   -66.332, E3 +150997.396}
SPL {X  -160.000, Y  +638.226, Z    +0.000, E1   -66.314, E3 +151012.724}
SPL {X  -160.000, Y  +655.092, Z    +0.000, E1   -66.336, E3 +151028.383}
SPL {X  -160.000, Y  +671.716, Z    +0.000, E1   -66.315, E3 +151043.897}
SPL {X  -159.502, Y  +687.017, Z    +0.000, E1   -66.266, E3 +151058.647}
SPL {X  -157.713, Y  +701.353, Z    +0.000, E1   -66.026, E3 +151073.874}
SPL {X  -155.081, Y  +713.767, Z    +0.000, E1   -65.665, E3 +151088.159}
SPL {X  -152.128, Y  +723.968, Z    +0.000, E1   -65.242, E3 +151100.659}
SPL {X  -148.925, Y  +732.892, Z    +0.000, E1   -64.779, E3 +151112.159}
SPL {X  -144.887, Y  +742.280, Z    +0.000, E1   -64.184, E3 +151124.788}
SPL {X  -140.317, Y  +751.285, Z    +0.000, E1   -63.454, E3 +151137.426}
SPL {X  -135.706, Y  +759.158, Z    +0.000, E1   -62.682, E3 +151148.827}
SPL {X  -131.040, Y  +766.207, Z    +0.000, E1   -61.854, E3 +151159.259}
SPL {X  -102.962, Y  +796.870, Z    +0.000, E1   -51.620, E3 +151284.591}
ENDSPLINE

SPLINE
SPL {X  -139.855, Y  +752.122, Z    +0.000, E1   -42.075, E3 +151407.519}
SPL {X  -153.268, Y  +720.324, Z    +0.000, E1   -30.648, E3 +151423.764}
SPL {X  -158.910, Y  +693.048, Z    +0.000, E1   -15.531, E3 +151429.835}
SPL {X  -159.977, Y  +677.095, Z    +0.000, E1    -3.968, E3 +151431.259}
SPL {X  -160.000, Y  +672.556, Z    +0.000, E1    -0.073, E3 +151431.361}
SPL {X  -160.000, Y  +669.399, Z    +0.000, E1    +3.976, E3 +151431.440}
SPL {X  -160.000, Y  +661.045, Z    +0.000, E1   +19.300, E3 +151432.029}
SPL {X  -160.000, Y  +646.999, Z    +0.000, E1   +41.048, E3 +151434.447}
SPL {X  -160.000, Y  +594.464, Z    +0.000, E1   +63.651, E3 +151454.747}
SPL {X  -160.000, Y  +465.200, Z    +0.000, E1   +67.027, E3 +151543.317}
SPL {X  -160.000, Y  +444.745, Z    +0.000, E1   +67.032, E3 +151561.726}
SPL {X  -160.000, Y  +422.224, Z    +0.000, E1   +67.044, E3 +151581.978}
ENDSPLINE

SPLINE
SPL {X  -160.000, Y  +424.635, Z    +0.000, E1   +64.425, E3 +151600.004}
ENDSPLINE

SPLINE
SPL {X  -160.000, Y  +410.501, Z    +0.000, E1   +64.162, E3 +151616.549}
SPL {X  -160.000, Y  +387.965, Z    +0.000, E1   +65.039, E3 +151632.500}
SPL {X  -158.836, Y  +366.435, Z    +0.000, E1   +65.805, E3 +151647.441}
SPL {X  -155.922, Y  +349.806, Z    +0.000, E1   +65.927, E3 +151662.088}
SPL {X  -152.875, Y  +338.486, Z    +0.000, E1   +65.488, E3 +151675.705}
SPL {X  -149.360, Y  +328.327, Z    +0.000, E1   +64.994, E3 +151688.611}
SPL {X  -145.195, Y  +318.481, Z    +0.000, E1   +64.365, E3 +151701.765}
SPL {X  -140.564, Y  +309.268, Z    +0.000, E1   +63.646, E3 +151714.586}
SPL {X  -135.770, Y  +301.044, Z    +0.000, E1   +62.840, E3 +151726.457}
SPL {X  -130.944, Y  +293.756, Z    +0.000, E1   +61.990, E3 +151737.200}
SPL {X  -103.957, Y  +264.074, Z    +0.000, E1   +52.557, E3 +151843.304}
ENDSPLINE

SPLINE
SPL {X  -133.093, Y  +296.896, Z    +0.000, E1   +44.059, E3 +151968.138}
SPL {X  -150.601, Y  +331.670, Z    +0.000, E1   +33.435, E3 +151992.400}
SPL {X  -157.739, Y  +358.898, Z    +0.000, E1   +20.026, E3 +152000.628}
SPL {X  -159.601, Y  +374.403, Z    +0.000, E1   +10.058, E3 +152002.944}
SPL {X  -159.993, Y  +384.251, Z    +0.000, E1    +2.830, E3 +152003.576}
SPL {X  -160.000, Y  +387.929, Z    +0.000, E1    -0.363, E3 +152003.644}
SPL {X  -160.000, Y  +392.137, Z    +0.000, E1    -6.580, E3 +152003.783}
SPL {X  -160.000, Y  +398.334, Z    +0.000, E1   -17.404, E3 +152004.275}
SPL {X  -160.000, Y  +410.558, Z    +0.000, E1   -36.649, E3 +152006.378}
SPL {X  -160.000, Y  +459.534, Z    +0.000, E1   -61.429, E3 +152025.972}
SPL {X  -160.000, Y  +586.246, Z    +0.000, E1   -66.315, E3 +152112.472}
SPL {X  -160.000, Y  +602.823, Z    +0.000, E1   -66.332, E3 +152127.876}
SPL {X  -160.000, Y  +621.796, Z    +0.000, E1   -66.332, E3 +152145.544}
SPL {X  -160.000, Y  +638.226, Z    +0.000, E1   -66.314, E3 +152160.872}
SPL {X  -160.000, Y  +655.092, Z    +0.000, E1   -66.336, E3 +152176.531}
SPL {X  -160.000, Y  +671.716, Z    +0.000, E1   -66.315, E3 +152192.045}
SPL {X  -159.502, Y  +687.017, Z    +0.000, E1   -66.266, E3 +152206.795}
SPL {X  -157.713, Y  +701.353, Z    +0.000, E1   -66.026, E3 +152222.022}
SPL {X  -155.081, Y  +713.767, Z    +0.000, E1   -65.665, E3 +152236.307}
SPL {X  -152.128, Y  +723.968, Z    +0.000, E1   -65.242, E3 +152248.807}
SPL {X  -148.925, Y  +732.892, Z    +0.000, E1   -64.779, E3 +152260.307}
SPL {X  -144.887, Y  +742.280, Z    +0.000, E1   -64.184, E3 +152272.936}
SPL {X  -140.317, Y  +751.285, Z    +0.000, E1   -63.454, E3 +152285.574}
SPL {X  -135.706, Y  +759.158, Z    +0.000, E1   -62.682, E3 +152296.975}
SPL {X  -131.040, Y  +766.207, Z    +0.000, E1   -61.854, E3 +152307.407}
SPL {X  -102.962, Y  +796.870, Z    +0.000, E1   -51.620, E3 +152432.738}
ENDSPLINE

SPLINE
SPL {X  -139.855, Y  +752.122, Z    +0.000, E1   -42.075, E3 +152555.667}
SPL {X  -153.268, Y  +720.324, Z    +0.000, E1   -30.648, E3 +152571.912}
SPL {X  -158.910, Y  +693.048, Z    +0.000, E1   -15.531, E3 +152577.983}
SPL {X  -159.977, Y  +677.095, Z    +0.000, E1    -3.968, E3 +152579.407}
SPL {X  -160.000, Y  +672.556, Z    +0.000, E1    -0.073, E3 +152579.509}
SPL {X  -160.000, Y  +669.399, Z    +0.000, E1    +3.976, E3 +152579.588}
SPL {X  -160.000, Y  +661.045, Z    +0.000, E1   +19.300, E3 +152580.177}
SPL {X  -160.000, Y  +646.999, Z    +0.000, E1   +41.048, E3 +152582.595}
SPL {X  -160.000, Y  +594.464, Z    +0.000, E1   +63.651, E3 +152602.895}
SPL {X  -160.000, Y  +465.200, Z    +0.000, E1   +67.027, E3 +152691.465}
SPL {X  -160.000, Y  +444.745, Z    +0.000, E1   +67.032, E3 +152709.874}
SPL {X  -160.000, Y  +422.224, Z    +0.000, E1   +67.044, E3 +152730.125}
ENDSPLINE

SPLINE
SPL {X  -160.000, Y  +424.635, Z    +0.000, E1   +64.425, E3 +152748.152}
ENDSPLINE

SPLINE
SPL {X  -160.000, Y  +410.501, Z    +0.000, E1   +64.162, E3 +152764.697}
SPL {X  -160.000, Y  +387.965, Z    +0.000, E1   +65.039, E3 +152780.648}
SPL {X  -158.836, Y  +366.435, Z    +0.000, E1   +65.805, E3 +152795.589}
SPL {X  -155.922, Y  +349.806, Z    +0.000, E1   +65.927, E3 +152810.236}
SPL {X  -152.875, Y  +338.486, Z    +0.000, E1   +65.488, E3 +152823.853}
SPL {X  -149.360, Y  +328.327, Z    +0.000, E1   +64.994, E3 +152836.759}
SPL {X  -145.195, Y  +318.481, Z    +0.000, E1   +64.365, E3 +152849.913}
SPL {X  -140.564, Y  +309.268, Z    +0.000, E1   +63.646, E3 +152862.734}
SPL {X  -135.770, Y  +301.044, Z    +0.000, E1   +62.840, E3 +152874.605}
SPL {X  -130.944, Y  +293.756, Z    +0.000, E1   +61.990, E3 +152885.348}
SPL {X  -103.957, Y  +264.074, Z    +0.000, E1   +52.557, E3 +152991.452}
ENDSPLINE

SPLINE
SPL {X  -133.093, Y  +296.896, Z    +0.000, E1   +44.059, E3 +153116.286}
SPL {X  -150.601, Y  +331.670, Z    +0.000, E1   +33.435, E3 +153140.548}
SPL {X  -157.739, Y  +358.898, Z    +0.000, E1   +20.026, E3 +153148.776}
SPL {X  -159.601, Y  +374.403, Z    +0.000, E1   +10.058, E3 +153151.092}
SPL {X  -159.993, Y  +384.251, Z    +0.000, E1    +2.830, E3 +153151.724}
SPL {X  -160.000, Y  +387.929, Z    +0.000, E1    -0.363, E3 +153151.792}
SPL {X  -160.000, Y  +392.137, Z    +0.000, E1    -6.580, E3 +153151.931}
SPL {X  -160.000, Y  +398.334, Z    +0.000, E1   -17.404, E3 +153152.423}
SPL {X  -160.000, Y  +410.558, Z    +0.000, E1   -36.649, E3 +153154.526}
SPL {X  -160.000, Y  +459.534, Z    +0.000, E1   -61.429, E3 +153174.120}
SPL {X  -160.000, Y  +586.246, Z    +0.000, E1   -66.315, E3 +153260.620}
SPL {X  -160.000, Y  +602.823, Z    +0.000, E1   -66.332, E3 +153276.024}
SPL {X  -160.000, Y  +621.796, Z    +0.000, E1   -66.332, E3 +153293.692}
SPL {X  -160.000, Y  +638.226, Z    +0.000, E1   -66.314, E3 +153309.020}
SPL {X  -160.000, Y  +655.092, Z    +0.000, E1   -66.336, E3 +153324.679}
SPL {X  -160.000, Y  +671.716, Z    +0.000, E1   -66.315, E3 +153340.192}
SPL {X  -159.502, Y  +687.017, Z    +0.000, E1   -66.266, E3 +153354.942}
SPL {X  -157.713, Y  +701.353, Z    +0.000, E1   -66.026, E3 +153370.170}
SPL {X  -155.081, Y  +713.767, Z    +0.000, E1   -65.665, E3 +153384.455}
SPL {X  -152.128, Y  +723.968, Z    +0.000, E1   -65.242, E3 +153396.955}
SPL {X  -148.925, Y  +732.892, Z    +0.000, E1   -64.779, E3 +153408.455}
SPL {X  -144.887, Y  +742.280, Z    +0.000, E1   -64.184, E3 +153421.084}
SPL {X  -140.317, Y  +751.285, Z    +0.000, E1   -63.454, E3 +153433.722}
SPL {X  -135.706, Y  +759.158, Z    +0.000, E1   -62.682, E3 +153445.123}
SPL {X  -131.040, Y  +766.207, Z    +0.000, E1   -61.854, E3 +153455.554}
SPL {X  -102.962, Y  +796.870, Z    +0.000, E1   -51.620, E3 +153580.886}
ENDSPLINE

SPLINE
SPL {X  -139.855, Y  +752.122, Z    +0.000, E1   -42.075, E3 +153703.815}
SPL {X  -153.268, Y  +720.324, Z    +0.000, E1   -30.648, E3 +153720.060}
SPL {X  -158.910, Y  +693.048, Z    +0.000, E1   -15.531, E3 +153726.131}
SPL {X  -159.977, Y  +677.095, Z    +0.000, E1    -3.968, E3 +153727.555}
SPL {X  -160.000, Y  +672.556, Z    +0.000, E1    -0.073, E3 +153727.657}
SPL {X  -160.000, Y  +669.399, Z    +0.000, E1    +3.976, E3 +153727.736}
SPL {X  -160.000, Y  +661.045, Z    +0.000, E1   +19.300, E3 +153728.325}
SPL {X  -160.000, Y  +646.999, Z    +0.000, E1   +41.048, E3 +153730.743}
SPL {X  -160.000, Y  +594.464, Z    +0.000, E1   +63.651, E3 +153751.043}
SPL {X  -160.000, Y  +465.200, Z    +0.000, E1   +67.027, E3 +153839.613}
SPL {X  -160.000, Y  +444.745, Z    +0.000, E1   +67.032, E3 +153858.022}
SPL {X  -160.000, Y  +422.224, Z    +0.000, E1   +67.044, E3 +153878.273}
ENDSPLINE

SPLINE
SPL {X  -160.000, Y  +424.635, Z    +0.000, E1   +64.425, E3 +153896.300}
ENDSPLINE

SPLINE
SPL {X  -160.000, Y  +410.501, Z    +0.000, E1   +64.162, E3 +153912.845}
SPL {X  -160.000, Y  +387.965, Z    +0.000, E1   +65.039, E3 +153928.796}
SPL {X  -158.836, Y  +366.435, Z    +0.000, E1   +65.805, E3 +153943.737}
SPL {X  -155.922, Y  +349.806, Z    +0.000, E1   +65.927, E3 +153958.384}
SPL {X  -152.875, Y  +338.486, Z    +0.000, E1   +65.488, E3 +153972.001}
SPL {X  -149.360, Y  +328.327, Z    +0.000, E1   +64.994, E3 +153984.907}
SPL {X  -145.195, Y  +318.481, Z    +0.000, E1   +64.365, E3 +153998.061}
SPL {X  -140.564, Y  +309.268, Z    +0.000, E1   +63.646, E3 +154010.882}
SPL {X  -135.770, Y  +301.044, Z    +0.000, E1   +62.840, E3 +154022.753}
SPL {X  -130.944, Y  +293.756, Z    +0.000, E1   +61.990, E3 +154033.496}
SPL {X  -103.957, Y  +264.074, Z    +0.000, E1   +52.557, E3 +154139.600}
ENDSPLINE

SPLINE
SPL {X  -133.093, Y  +296.896, Z    +0.000, E1   +44.059, E3 +154264.434}
SPL {X  -150.601, Y  +331.670, Z    +0.000, E1   +33.435, E3 +154288.696}
SPL {X  -157.739, Y  +358.898, Z    +0.000, E1   +20.026, E3 +154296.924}
SPL {X  -159.601, Y  +374.403, Z    +0.000, E1   +10.058, E3 +154299.240}
SPL {X  -159.993, Y  +384.251, Z    +0.000, E1    +2.830, E3 +154299.872}
SPL {X  -160.000, Y  +387.929, Z    +0.000, E1    -0.363, E3 +154299.940}
SPL {X  -160.000, Y  +392.137, Z    +0.000, E1    -6.580, E3 +154300.079}
SPL {X  -160.000, Y  +398.334, Z    +0.000, E1   -17.404, E3 +154300.571}
SPL {X  -160.000, Y  +410.558, Z    +0.000, E1   -36.649, E3 +154302.674}
SPL {X  -160.000, Y  +459.534, Z    +0.000, E1   -61.429, E3 +154322.268}
SPL {X  -160.000, Y  +586.246, Z    +0.000, E1   -66.315, E3 +154408.768}
SPL {X  -160.000, Y  +602.823, Z    +0.000, E1   -66.332, E3 +154424.172}
SPL {X  -160.000, Y  +621.796, Z    +0.000, E1   -66.332, E3 +154441.840}
SPL {X  -160.000, Y  +638.226, Z    +0.000, E1   -66.314, E3 +154457.168}
SPL {X  -160.000, Y  +655.092, Z    +0.000, E1   -66.336, E3 +154472.826}
SPL {X  -160.000, Y  +671.716, Z    +0.000, E1   -66.315, E3 +154488.340}
SPL {X  -159.502, Y  +687.017, Z    +0.000, E1   -66.266, E3 +154503.090}
SPL {X  -157.713, Y  +701.353, Z    +0.000, E1   -66.026, E3 +154518.318}
SPL {X  -155.081, Y  +713.767, Z    +0.000, E1   -65.665, E3 +154532.603}
SPL {X  -152.128, Y  +723.968, Z    +0.000, E1   -65.242, E3 +154545.103}
SPL {X  -148.925, Y  +732.892, Z    +0.000, E1   -64.779, E3 +154556.603}
SPL {X  -144.887, Y  +742.280, Z    +0.000, E1   -64.184, E3 +154569.232}
SPL {X  -140.317, Y  +751.285, Z    +0.000, E1   -63.454, E3 +154581.870}
SPL {X  -135.706, Y  +759.158, Z    +0.000, E1   -62.682, E3 +154593.271}
SPL {X  -131.040, Y  +766.207, Z    +0.000, E1   -61.854, E3 +154603.702}
SPL {X  -102.962, Y  +796.870, Z    +0.000, E1   -51.620, E3 +154729.034}
ENDSPLINE

SPLINE
SPL {X  -139.855, Y  +752.122, Z    +0.000, E1   -42.075, E3 +154851.963}
SPL {X  -153.268, Y  +720.324, Z    +0.000, E1   -30.648, E3 +154868.208}
SPL {X  -158.910, Y  +693.048, Z    +0.000, E1   -15.531, E3 +154874.279}
SPL {X  -159.977, Y  +677.095, Z    +0.000, E1    -3.968, E3 +154875.703}
SPL {X  -160.000, Y  +672.556, Z    +0.000, E1    -0.073, E3 +154875.805}
SPL {X  -160.000, Y  +669.399, Z    +0.000, E1    +3.976, E3 +154875.884}
SPL {X  -160.000, Y  +661.045, Z    +0.000, E1   +19.300, E3 +154876.473}
SPL {X  -160.000, Y  +646.999, Z    +0.000, E1   +41.048, E3 +154878.891}
SPL {X  -160.000, Y  +594.464, Z    +0.000, E1   +63.651, E3 +154899.191}
SPL {X  -160.000, Y  +465.200, Z    +0.000, E1   +67.027, E3 +154987.761}
SPL {X  -160.000, Y  +444.745, Z    +0.000, E1   +67.032, E3 +155006.170}
SPL {X  -160.000, Y  +422.224, Z    +0.000, E1   +67.044, E3 +155026.421}
ENDSPLINE

SPLINE
SPL {X  -160.000, Y  +424.635, Z    +0.000, E1   +64.425, E3 +155044.448}
ENDSPLINE

SPLINE
SPL {X  -160.000, Y  +410.501, Z    +0.000, E1   +64.162, E3 +155060.993}
SPL {X  -160.000, Y  +387.965, Z    +0.000, E1   +65.039, E3 +155076.944}
SPL {X  -158.836, Y  +366.435, Z    +0.000, E1   +65.805, E3 +155091.885}
SPL {X  -155.922, Y  +349.806, Z    +0.000, E1   +65.927, E3 +155106.532}
SPL {X  -152.875, Y  +338.486, Z    +0.000, E1   +65.488, E3 +155120.149}
SPL {X  -149.360, Y  +328.327, Z    +0.000, E1   +64.994, E3 +155133.055}
SPL {X  -145.195, Y  +318.481, Z    +0.000, E1   +64.365, E3 +155146.209}
SPL {X  -140.564, Y  +309.268, Z    +0.000, E1   +63.646, E3 +155159.030}
SPL {X  -135.770, Y  +301.044, Z    +0.000, E1   +62.840, E3 +155170.901}
SPL {X  -130.944, Y  +293.756, Z    +0.000, E1   +61.990, E3 +155181.644}
SPL {X  -103.957, Y  +264.074, Z    +0.000, E1   +52.557, E3 +155287.748}
ENDSPLINE

SPLINE
SPL {X  -133.093, Y  +296.896, Z    +0.000, E1   +44.059, E3 +155412.582}
SPL {X  -150.601, Y  +331.670, Z    +0.000, E1   +33.435, E3 +155436.844}
SPL {X  -157.739, Y  +358.898, Z    +0.000, E1   +20.026, E3 +155445.072}
SPL {X  -159.601, Y  +374.403, Z    +0.000, E1   +10.058, E3 +155447.388}
SPL {X  -159.993, Y  +384.251, Z    +0.000, E1    +2.830, E3 +155448.020}
SPL {X  -160.000, Y  +387.929, Z    +0.000, E1    -0.363, E3 +155448.088}
SPL {X  -160.000, Y  +392.137, Z    +0.000, E1    -6.580, E3 +155448.227}
SPL {X  -160.000, Y  +398.334, Z    +0.000, E1   -17.404, E3 +155448.719}
SPL {X  -160.000, Y  +410.558, Z    +0.000, E1   -36.649, E3 +155450.822}
SPL {X  -160.000, Y  +459.534, Z    +0.000, E1   -61.429, E3 +155470.416}
SPL {X  -160.000, Y  +586.246, Z    +0.000, E1   -66.315, E3 +155556.916}
SPL {X  -160.000, Y  +602.823, Z    +0.000, E1   -66.332, E3 +155572.320}
SPL {X  -160.000, Y  +621.796, Z    +0.000, E1   -66.332, E3 +155589.988}
SPL {X  -160.000, Y  +638.226, Z    +0.000, E1   -66.314, E3 +155605.316}
SPL {X  -160.000, Y  +655.092, Z    +0.000, E1   -66.336, E3 +155620.974}
SPL {X  -160.000, Y  +671.716, Z    +0.000, E1   -66.315, E3 +155636.488}
SPL {X  -159.502, Y  +687.017, Z    +0.000, E1   -66.266, E3 +155651.238}
SPL {X  -157.713, Y  +701.353, Z    +0.000, E1   -66.026, E3 +155666.466}
SPL {X  -155.081, Y  +713.767, Z    +0.000, E1   -65.665, E3 +155680.751}
SPL {X  -152.128, Y  +723.968, Z    +0.000, E1   -65.242, E3 +155693.251}
SPL {X  -148.925, Y  +732.892, Z    +0.000, E1   -64.779, E3 +155704.750}
SPL {X  -144.887, Y  +742.280, Z    +0.000, E1   -64.184, E3 +155717.380}
SPL {X  -140.317, Y  +751.285, Z    +0.000, E1   -63.454, E3 +155730.018}
SPL {X  -135.706, Y  +759.158, Z    +0.000, E1   -62.682, E3 +155741.419}
SPL {X  -131.040, Y  +766.207, Z    +0.000, E1   -61.854, E3 +155751.850}
SPL {X  -102.962, Y  +796.870, Z    +0.000, E1   -51.620, E3 +155877.182}
ENDSPLINE

SPLINE
SPL {X  -139.855, Y  +752.122, Z    +0.000, E1   -42.075, E3 +156000.111}
SPL {X  -153.268, Y  +720.324, Z    +0.000, E1   -30.648, E3 +156016.356}
SPL {X  -158.910, Y  +693.048, Z    +0.000, E1   -15.531, E3 +156022.427}
SPL {X  -159.977, Y  +677.095, Z    +0.000, E1    -3.968, E3 +156023.851}
SPL {X  -160.000, Y  +672.556, Z    +0.000, E1    -0.073, E3 +156023.953}
SPL {X  -160.000, Y  +669.399, Z    +0.000, E1    +3.976, E3 +156024.032}
SPL {X  -160.000, Y  +661.045, Z    +0.000, E1   +19.300, E3 +156024.621}
SPL {X  -160.000, Y  +646.999, Z    +0.000, E1   +41.048, E3 +156027.038}
SPL {X  -160.000, Y  +594.464, Z    +0.000, E1   +63.651, E3 +156047.339}
SPL {X  -160.000, Y  +465.200, Z    +0.000, E1   +67.027, E3 +156135.909}
SPL {X  -160.000, Y  +444.745, Z    +0.000, E1   +67.032, E3 +156154.318}
SPL {X  -160.000, Y  +422.224, Z    +0.000, E1   +67.044, E3 +156174.569}
ENDSPLINE

SPLINE
SPL {X  -160.000, Y  +424.635, Z    +0.000, E1   +64.425, E3 +156192.596}
ENDSPLINE

SPLINE
SPL {X  -160.000, Y  +410.501, Z    +0.000, E1   +64.162, E3 +156209.141}
SPL {X  -160.000, Y  +387.965, Z    +0.000, E1   +65.039, E3 +156225.092}
SPL {X  -158.836, Y  +366.435, Z    +0.000, E1   +65.805, E3 +156240.033}
SPL {X  -155.922, Y  +349.806, Z    +0.000, E1   +65.927, E3 +156254.680}
SPL {X  -152.875, Y  +338.486, Z    +0.000, E1   +65.488, E3 +156268.297}
SPL {X  -149.360, Y  +328.327, Z    +0.000, E1   +64.994, E3 +156281.203}
SPL {X  -145.195, Y  +318.481, Z    +0.000, E1   +64.365, E3 +156294.357}
SPL {X  -140.564, Y  +309.268, Z    +0.000, E1   +63.646, E3 +156307.178}
SPL {X  -135.770, Y  +301.044, Z    +0.000, E1   +62.840, E3 +156319.049}
SPL {X  -130.944, Y  +293.756, Z    +0.000, E1   +61.990, E3 +156329.792}
SPL {X  -103.957, Y  +264.074, Z    +0.000, E1   +52.557, E3 +156435.896}
ENDSPLINE

SPLINE
SPL {X  -133.093, Y  +296.896, Z    +0.000, E1   +44.059, E3 +156560.730}
SPL {X  -150.601, Y  +331.670, Z    +0.000, E1   +33.435, E3 +156584.992}
SPL {X  -157.739, Y  +358.898, Z    +0.000, E1   +20.026, E3 +156593.220}
SPL {X  -159.601, Y  +374.403, Z    +0.000, E1   +10.058, E3 +156595.536}
SPL {X  -159.993, Y  +384.251, Z    +0.000, E1    +2.830, E3 +156596.168}
SPL {X  -160.000, Y  +387.929, Z    +0.000, E1    -0.363, E3 +156596.236}
SPL {X  -160.000, Y  +392.137, Z    +0.000, E1    -6.580, E3 +156596.375}
SPL {X  -160.000, Y  +398.334, Z    +0.000, E1   -17.404, E3 +156596.867}
SPL {X  -160.000, Y  +410.558, Z    +0.000, E1   -36.649, E3 +156598.969}
SPL {X  -160.000, Y  +459.534, Z    +0.000, E1   -61.429, E3 +156618.564}
SPL {X  -160.000, Y  +586.246, Z    +0.000, E1   -66.315, E3 +156705.064}
SPL {X  -160.000, Y  +602.823, Z    +0.000, E1   -66.332, E3 +156720.468}
SPL {X  -160.000, Y  +621.796, Z    +0.000, E1   -66.332, E3 +156738.136}
SPL {X  -160.000, Y  +638.226, Z    +0.000, E1   -66.314, E3 +156753.464}
SPL {X  -160.000, Y  +655.092, Z    +0.000, E1   -66.336, E3 +156769.122}
SPL {X  -160.000, Y  +671.716, Z    +0.000, E1   -66.315, E3 +156784.636}
SPL {X  -159.502, Y  +687.017, Z    +0.000, E1   -66.266, E3 +156799.386}
SPL {X  -157.713, Y  +701.353, Z    +0.000, E1   -66.026, E3 +156814.614}
SPL {X  -155.081, Y  +713.767, Z    +0.000, E1   -65.665, E3 +156828.899}
SPL {X  -152.128, Y  +723.968, Z    +0.000, E1   -65.242, E3 +156841.399}
SPL {X  -148.925, Y  +732.892, Z    +0.000, E1   -64.779, E3 +156852.898}
SPL {X  -144.887, Y  +742.280, Z    +0.000, E1   -64.184, E3 +156865.528}
SPL {X  -140.317, Y  +751.285, Z    +0.000, E1   -63.454, E3 +156878.166}
SPL {X  -135.706, Y  +759.158, Z    +0.000, E1   -62.682, E3 +156889.567}
SPL {X  -131.040, Y  +766.207, Z    +0.000, E1   -61.854, E3 +156899.998}
SPL {X  -102.962, Y  +796.870, Z    +0.000, E1   -51.620, E3 +157025.330}
ENDSPLINE

SPLINE
SPL {X  -139.855, Y  +752.122, Z    +0.000, E1   -42.075, E3 +157148.259}
SPL {X  -153.268, Y  +720.324, Z    +0.000, E1   -30.648, E3 +157164.504}
SPL {X  -158.910, Y  +693.048, Z    +0.000, E1   -15.531, E3 +157170.575}
SPL {X  -159.977, Y  +677.095, Z    +0.000, E1    -3.968, E3 +157171.999}
SPL {X  -160.000, Y  +672.556, Z    +0.000, E1    -0.073, E3 +157172.101}
SPL {X  -160.000, Y  +669.399, Z    +0.000, E1    +3.976, E3 +157172.180}
SPL {X  -160.000, Y  +661.045, Z    +0.000, E1   +19.300, E3 +157172.769}
SPL {X  -160.000, Y  +646.999, Z    +0.000, E1   +41.048, E3 +157175.186}
SPL {X  -160.000, Y  +594.464, Z    +0.000, E1   +63.651, E3 +157195.487}
SPL {X  -160.000, Y  +465.200, Z    +0.000, E1   +67.027, E3 +157284.057}
SPL {X  -160.000, Y  +444.745, Z    +0.000, E1   +67.032, E3 +157302.466}
SPL {X  -160.000, Y  +422.224, Z    +0.000, E1   +67.044, E3 +157322.717}
ENDSPLINE

SPLINE
SPL {X  -160.000, Y  +424.635, Z    +0.000, E1   +64.425, E3 +157340.744}
ENDSPLINE

SPLINE
SPL {X  -160.000, Y  +410.501, Z    +0.000, E1   +64.162, E3 +157357.289}
SPL {X  -160.000, Y  +387.965, Z    +0.000, E1   +65.039, E3 +157373.240}
SPL {X  -158.836, Y  +366.435, Z    +0.000, E1   +65.805, E3 +157388.181}
SPL {X  -155.922, Y  +349.806, Z    +0.000, E1   +65.927, E3 +157402.828}
SPL {X  -152.875, Y  +338.486, Z    +0.000, E1   +65.488, E3 +157416.445}
SPL {X  -149.360, Y  +328.327, Z    +0.000, E1   +64.994, E3 +157429.351}
SPL {X  -145.195, Y  +318.481, Z    +0.000, E1   +64.365, E3 +157442.505}
SPL {X  -140.564, Y  +309.268, Z    +0.000, E1   +63.646, E3 +157455.326}
SPL {X  -135.770, Y  +301.044, Z    +0.000, E1   +62.840, E3 +157467.197}
SPL {X  -130.944, Y  +293.756, Z    +0.000, E1   +61.990, E3 +157477.940}
SPL {X  -103.957, Y  +264.074, Z    +0.000, E1   +52.557, E3 +157584.044}
ENDSPLINE

SPLINE
SPL {X  -133.093, Y  +296.896, Z    +0.000, E1   +44.059, E3 +157708.878}
SPL {X  -150.601, Y  +331.670, Z    +0.000, E1   +33.435, E3 +157733.140}
SPL {X  -157.739, Y  +358.898, Z    +0.000, E1   +20.026, E3 +157741.368}
SPL {X  -159.601, Y  +374.403, Z    +0.000, E1   +10.058, E3 +157743.684}
SPL {X  -159.993, Y  +384.251, Z    +0.000, E1    +2.830, E3 +157744.316}
SPL {X  -160.000, Y  +387.929, Z    +0.000, E1    -0.363, E3 +157744.384}
SPL {X  -160.000, Y  +392.137, Z    +0.000, E1    -6.580, E3 +157744.523}
SPL {X  -160.000, Y  +398.334, Z    +0.000, E1   -17.404, E3 +157745.015}
SPL {X  -160.000, Y  +410.558, Z    +0.000, E1   -36.649, E3 +157747.117}
SPL {X  -160.000, Y  +459.534, Z    +0.000, E1   -61.429, E3 +157766.712}
SPL {X  -160.000, Y  +586.246, Z    +0.000, E1   -66.315, E3 +157853.212}
SPL {X  -160.000, Y  +602.823, Z    +0.000, E1   -66.332, E3 +157868.616}
SPL {X  -160.000, Y  +621.796, Z    +0.000, E1   -66.332, E3 +157886.284}
SPL {X  -160.000, Y  +638.226, Z    +0.000, E1   -66.314, E3 +157901.612}
SPL {X  -160.000, Y  +655.092, Z    +0.000, E1   -66.336, E3 +157917.270}
SPL {X  -160.000, Y  +671.716, Z    +0.000, E1   -66.315, E3 +157932.784}
SPL {X  -159.502, Y  +687.017, Z    +0.000, E1   -66.266, E3 +157947.534}
SPL {X  -157.713, Y  +701.353, Z    +0.000, E1   -66.026, E3 +157962.762}
SPL {X  -155.081, Y  +713.767, Z    +0.000, E1   -65.665, E3 +157977.047}
SPL {X  -152.128, Y  +723.968, Z    +0.000, E1   -65.242, E3 +157989.546}
SPL {X  -148.925, Y  +732.892, Z    +0.000, E1   -64.779, E3 +158001.046}
SPL {X  -144.887, Y  +742.280, Z    +0.000, E1   -64.184, E3 +158013.676}
SPL {X  -140.317, Y  +751.285, Z    +0.000, E1   -63.454, E3 +158026.314}
SPL {X  -135.706, Y  +759.158, Z    +0.000, E1   -62.682, E3 +158037.715}
SPL {X  -131.040, Y  +766.207, Z    +0.000, E1   -61.854, E3 +158048.146}
SPL {X  -102.962, Y  +796.870, Z    +0.000, E1   -51.620, E3 +158173.478}
ENDSPLINE

SPLINE
SPL {X  -139.855, Y  +752.122, Z    +0.000, E1   -42.075, E3 +158296.407}
SPL {X  -153.268, Y  +720.324, Z    +0.000, E1   -30.648, E3 +158312.652}
SPL {X  -158.910, Y  +693.048, Z    +0.000, E1   -15.531, E3 +158318.723}
SPL {X  -159.977, Y  +677.095, Z    +0.000, E1    -3.968, E3 +158320.147}
SPL {X  -160.000, Y  +672.556, Z    +0.000, E1    -0.073, E3 +158320.249}
SPL {X  -160.000, Y  +669.399, Z    +0.000, E1    +3.976, E3 +158320.328}
SPL {X  -160.000, Y  +661.045, Z    +0.000, E1   +19.300, E3 +158320.917}
SPL {X  -160.000, Y  +646.999, Z    +0.000, E1   +41.048, E3 +158323.334}
SPL {X  -160.000, Y  +594.464, Z    +0.000, E1   +63.651, E3 +158343.635}
SPL {X  -160.000, Y  +465.200, Z    +0.000, E1   +67.027, E3 +158432.205}
SPL {X  -160.000, Y  +444.745, Z    +0.000, E1   +67.032, E3 +158450.614}
SPL {X  -160.000, Y  +422.224, Z    +0.000, E1   +67.044, E3 +158470.865}
ENDSPLINE

SPLINE
SPL {X  -160.000, Y  +424.635, Z    +0.000, E1   +64.425, E3 +158488.892}
ENDSPLINE

SPLINE
SPL {X  -160.000, Y  +410.501, Z    +0.000, E1   +64.162, E3 +158505.437}
SPL {X  -160.000, Y  +387.965, Z    +0.000, E1   +65.039, E3 +158521.388}
SPL {X  -158.836, Y  +366.435, Z    +0.000, E1   +65.805, E3 +158536.329}
SPL {X  -155.922, Y  +349.806, Z    +0.000, E1   +65.927, E3 +158550.976}
SPL {X  -152.875, Y  +338.486, Z    +0.000, E1   +65.488, E3 +158564.593}
SPL {X  -149.360, Y  +328.327, Z    +0.000, E1   +64.994, E3 +158577.499}
SPL {X  -145.195, Y  +318.481, Z    +0.000, E1   +64.365, E3 +158590.653}
SPL {X  -140.564, Y  +309.268, Z    +0.000, E1   +63.646, E3 +158603.474}
SPL {X  -135.770, Y  +301.044, Z    +0.000, E1   +62.840, E3 +158615.345}
SPL {X  -130.944, Y  +293.756, Z    +0.000, E1   +61.990, E3 +158626.088}
SPL {X  -103.957, Y  +264.074, Z    +0.000, E1   +52.557, E3 +158732.192}
ENDSPLINE

SPLINE
SPL {X  -133.093, Y  +296.896, Z    +0.000, E1   +44.059, E3 +158857.025}
SPL {X  -150.601, Y  +331.670, Z    +0.000, E1   +33.435, E3 +158881.288}
SPL {X  -157.739, Y  +358.898, Z    +0.000, E1   +20.026, E3 +158889.516}
SPL {X  -159.601, Y  +374.403, Z    +0.000, E1   +10.058, E3 +158891.832}
SPL {X  -159.993, Y  +384.251, Z    +0.000, E1    +2.830, E3 +158892.464}
SPL {X  -160.000, Y  +387.929, Z    +0.000, E1    -0.363, E3 +158892.532}
SPL {X  -160.000, Y  +392.137, Z    +0.000, E1    -6.580, E3 +158892.671}
SPL {X  -160.000, Y  +398.334, Z    +0.000, E1   -17.404, E3 +158893.163}
SPL {X  -160.000, Y  +410.558, Z    +0.000, E1   -36.649, E3 +158895.265}
SPL {X  -160.000, Y  +459.534, Z    +0.000, E1   -61.429, E3 +158914.860}
SPL {X  -160.000, Y  +586.246, Z    +0.000, E1   -66.315, E3 +159001.360}
SPL {X  -160.000, Y  +602.823, Z    +0.000, E1   -66.332, E3 +159016.764}
SPL {X  -160.000, Y  +621.796, Z    +0.000, E1   -66.332, E3 +159034.432}
SPL {X  -160.000, Y  +638.226, Z    +0.000, E1   -66.314, E3 +159049.760}
SPL {X  -160.000, Y  +655.092, Z    +0.000, E1   -66.336, E3 +159065.418}
SPL {X  -160.000, Y  +671.716, Z    +0.000, E1   -66.315, E3 +159080.932}
SPL {X  -159.502, Y  +687.017, Z    +0.000, E1   -66.266, E3 +159095.682}
SPL {X  -157.713, Y  +701.353, Z    +0.000, E1   -66.026, E3 +159110.910}
SPL {X  -155.081, Y  +713.767, Z    +0.000, E1   -65.665, E3 +159125.195}
SPL {X  -152.128, Y  +723.968, Z    +0.000, E1   -65.242, E3 +159137.694}
SPL {X  -148.925, Y  +732.892, Z    +0.000, E1   -64.779, E3 +159149.194}
SPL {X  -144.887, Y  +742.280, Z    +0.000, E1   -64.184, E3 +159161.824}
SPL {X  -140.317, Y  +751.285, Z    +0.000, E1   -63.454, E3 +159174.461}
SPL {X  -135.706, Y  +759.158, Z    +0.000, E1   -62.682, E3 +159185.863}
SPL {X  -131.040, Y  +766.207, Z    +0.000, E1   -61.854, E3 +159196.294}
SPL {X  -102.962, Y  +796.870, Z    +0.000, E1   -51.620, E3 +159321.626}
ENDSPLINE

SPLINE
SPL {X  -139.855, Y  +752.122, Z    +0.000, E1   -42.075, E3 +159444.555}
SPL {X  -153.268, Y  +720.324, Z    +0.000, E1   -30.648, E3 +159460.800}
SPL {X  -158.910, Y  +693.048, Z    +0.000, E1   -15.531, E3 +159466.871}
SPL {X  -159.977, Y  +677.095, Z    +0.000, E1    -3.968, E3 +159468.295}
SPL {X  -160.000, Y  +672.556, Z    +0.000, E1    -0.073, E3 +159468.397}
SPL {X  -160.000, Y  +669.399, Z    +0.000, E1    +3.976, E3 +159468.476}
SPL {X  -160.000, Y  +661.045, Z    +0.000, E1   +19.300, E3 +159469.065}
SPL {X  -160.000, Y  +646.999, Z    +0.000, E1   +41.048, E3 +159471.482}
SPL {X  -160.000, Y  +594.464, Z    +0.000, E1   +63.651, E3 +159491.783}
SPL {X  -160.000, Y  +465.200, Z    +0.000, E1   +67.027, E3 +159580.353}
SPL {X  -160.000, Y  +444.745, Z    +0.000, E1   +67.032, E3 +159598.762}
SPL {X  -160.000, Y  +422.224, Z    +0.000, E1   +67.044, E3 +159619.013}
ENDSPLINE

SPLINE
SPL {X  -160.000, Y  +424.635, Z    +0.000, E1   +64.425, E3 +159637.040}
ENDSPLINE

SPLINE
SPL {X  -160.000, Y  +410.501, Z    +0.000, E1   +64.162, E3 +159653.585}
SPL {X  -160.000, Y  +387.965, Z    +0.000, E1   +65.039, E3 +159669.536}
SPL {X  -158.836, Y  +366.435, Z    +0.000, E1   +65.805, E3 +159684.477}
SPL {X  -155.922, Y  +349.806, Z    +0.000, E1   +65.927, E3 +159699.124}
SPL {X  -152.875, Y  +338.486, Z    +0.000, E1   +65.488, E3 +159712.740}
SPL {X  -149.360, Y  +328.327, Z    +0.000, E1   +64.994, E3 +159725.647}
SPL {X  -145.195, Y  +318.481, Z    +0.000, E1   +64.365, E3 +159738.801}
SPL {X  -140.564, Y  +309.268, Z    +0.000, E1   +63.646, E3 +159751.622}
SPL {X  -135.770, Y  +301.044, Z    +0.000, E1   +62.840, E3 +159763.493}
SPL {X  -130.944, Y  +293.756, Z    +0.000, E1   +61.990, E3 +159774.236}
SPL {X  -103.957, Y  +264.074, Z    +0.000, E1   +52.557, E3 +159880.340}
ENDSPLINE

SPLINE
SPL {X  -133.093, Y  +296.896, Z    +0.000, E1   +44.059, E3 +160005.173}
SPL {X  -150.601, Y  +331.670, Z    +0.000, E1   +33.435, E3 +160029.436}
SPL {X  -157.739, Y  +358.898, Z    +0.000, E1   +20.026, E3 +160037.664}
SPL {X  -159.601, Y  +374.403, Z    +0.000, E1   +10.058, E3 +160039.979}
SPL {X  -159.993, Y  +384.251, Z    +0.000, E1    +2.830, E3 +160040.612}
SPL {X  -160.000, Y  +387.929, Z    +0.000, E1    -0.363, E3 +160040.680}
SPL {X  -160.000, Y  +392.137, Z    +0.000, E1    -6.580, E3 +160040.819}
SPL {X  -160.000, Y  +398.334, Z    +0.000, E1   -17.404, E3 +160041.311}
SPL {X  -160.000, Y  +410.558, Z    +0.000, E1   -36.649, E3 +160043.413}
SPL {X  -160.000, Y  +459.534, Z    +0.000, E1   -61.429, E3 +160063.008}
SPL {X  -160.000, Y  +586.246, Z    +0.000, E1   -66.315, E3 +160149.508}
SPL {X  -160.000, Y  +602.823, Z    +0.000, E1   -66.332, E3 +160164.912}
SPL {X  -160.000, Y  +621.796, Z    +0.000, E1   -66.332, E3 +160182.580}
SPL {X  -160.000, Y  +638.226, Z    +0.000, E1   -66.314, E3 +160197.908}
SPL {X  -160.000, Y  +655.092, Z    +0.000, E1   -66.336, E3 +160213.566}
SPL {X  -160.000, Y  +671.716, Z    +0.000, E1   -66.315, E3 +160229.080}
SPL {X  -159.502, Y  +687.017, Z    +0.000, E1   -66.266, E3 +160243.830}
SPL {X  -157.713, Y  +701.353, Z    +0.000, E1   -66.026, E3 +160259.058}
SPL {X  -155.081, Y  +713.767, Z    +0.000, E1   -65.665, E3 +160273.343}
SPL {X  -152.128, Y  +723.968, Z    +0.000, E1   -65.242, E3 +160285.842}
SPL {X  -148.925, Y  +732.892, Z    +0.000, E1   -64.779, E3 +160297.342}
SPL {X  -144.887, Y  +742.280, Z    +0.000, E1   -64.184, E3 +160309.972}
SPL {X  -140.317, Y  +751.285, Z    +0.000, E1   -63.454, E3 +160322.609}
SPL {X  -135.706, Y  +759.158, Z    +0.000, E1   -62.682, E3 +160334.011}
SPL {X  -131.040, Y  +766.207, Z    +0.000, E1   -61.854, E3 +160344.442}
SPL {X  -102.962, Y  +796.870, Z    +0.000, E1   -51.620, E3 +160469.774}
ENDSPLINE

SPLINE
SPL {X  -139.855, Y  +752.122, Z    +0.000, E1   -42.075, E3 +160592.703}
SPL {X  -153.268, Y  +720.324, Z    +0.000, E1   -30.648, E3 +160608.948}
SPL {X  -158.910, Y  +693.048, Z    +0.000, E1   -15.531, E3 +160615.019}
SPL {X  -159.977, Y  +677.095, Z    +0.000, E1    -3.968, E3 +160616.442}
SPL {X  -160.000, Y  +672.556, Z    +0.000, E1    -0.073, E3 +160616.545}
SPL {X  -160.000, Y  +669.399, Z    +0.000, E1    +3.976, E3 +160616.624}
SPL {X  -160.000, Y  +661.045, Z    +0.000, E1   +19.300, E3 +160617.213}
SPL {X  -160.000, Y  +646.999, Z    +0.000, E1   +41.048, E3 +160619.630}
SPL {X  -160.000, Y  +594.464, Z    +0.000, E1   +63.651, E3 +160639.931}
SPL {X  -160.000, Y  +465.200, Z    +0.000, E1   +67.027, E3 +160728.501}
SPL {X  -160.000, Y  +444.745, Z    +0.000, E1   +67.032, E3 +160746.910}
SPL {X  -160.000, Y  +422.224, Z    +0.000, E1   +67.044, E3 +160767.161}
ENDSPLINE

SPLINE
SPL {X  -160.000, Y  +424.635, Z    +0.000, E1   +64.425, E3 +160785.188}
ENDSPLINE

SPLINE
SPL {X  -160.000, Y  +410.501, Z    +0.000, E1   +64.162, E3 +160801.732}
SPL {X  -160.000, Y  +387.965, Z    +0.000, E1   +65.039, E3 +160817.684}
SPL {X  -158.836, Y  +366.435, Z    +0.000, E1   +65.805, E3 +160832.625}
SPL {X  -155.922, Y  +349.806, Z    +0.000, E1   +65.927, E3 +160847.272}
SPL {X  -152.875, Y  +338.486, Z    +0.000, E1   +65.488, E3 +160860.888}
SPL {X  -149.360, Y  +328.327, Z    +0.000, E1   +64.994, E3 +160873.795}
SPL {X  -145.195, Y  +318.481, Z    +0.000, E1   +64.365, E3 +160886.949}
SPL {X  -140.564, Y  +309.268, Z    +0.000, E1   +63.646, E3 +160899.769}
SPL {X  -135.770, Y  +301.044, Z    +0.000, E1   +62.840, E3 +160911.641}
SPL {X  -130.944, Y  +293.756, Z    +0.000, E1   +61.990, E3 +160922.384}
SPL {X  -103.957, Y  +264.074, Z    +0.000, E1   +52.557, E3 +161028.488}
ENDSPLINE

SPLINE
SPL {X  -133.093, Y  +296.896, Z    +0.000, E1   +44.059, E3 +161153.321}
SPL {X  -150.601, Y  +331.670, Z    +0.000, E1   +33.435, E3 +161177.584}
SPL {X  -157.739, Y  +358.898, Z    +0.000, E1   +20.026, E3 +161185.812}
SPL {X  -159.601, Y  +374.403, Z    +0.000, E1   +10.058, E3 +161188.127}
SPL {X  -159.993, Y  +384.251, Z    +0.000, E1    +2.830, E3 +161188.759}
SPL {X  -160.000, Y  +387.929, Z    +0.000, E1    -0.363, E3 +161188.828}
SPL {X  -160.000, Y  +392.137, Z    +0.000, E1    -6.580, E3 +161188.967}
SPL {X  -160.000, Y  +398.334, Z    +0.000, E1   -17.404, E3 +161189.459}
SPL {X  -160.000, Y  +410.558, Z    +0.000, E1   -36.649, E3 +161191.561}
SPL {X  -160.000, Y  +459.534, Z    +0.000, E1   -61.429, E3 +161211.156}
SPL {X  -160.000, Y  +586.246, Z    +0.000, E1   -66.315, E3 +161297.656}
SPL {X  -160.000, Y  +602.823, Z    +0.000, E1   -66.332, E3 +161313.060}
SPL {X  -160.000, Y  +621.796, Z    +0.000, E1   -66.332, E3 +161330.728}
SPL {X  -160.000, Y  +638.226, Z    +0.000, E1   -66.314, E3 +161346.056}
SPL {X  -160.000, Y  +655.092, Z    +0.000, E1   -66.336, E3 +161361.714}
SPL {X  -160.000, Y  +671.716, Z    +0.000, E1   -66.315, E3 +161377.228}
SPL {X  -159.502, Y  +687.017, Z    +0.000, E1   -66.266, E3 +161391.978}
SPL {X  -157.713, Y  +701.353, Z    +0.000, E1   -66.026, E3 +161407.205}
SPL {X  -155.081, Y  +713.767, Z    +0.000, E1   -65.665, E3 +161421.491}
SPL {X  -152.128, Y  +723.968, Z    +0.000, E1   -65.242, E3 +161433.990}
SPL {X  -148.925, Y  +732.892, Z    +0.000, E1   -64.779, E3 +161445.490}
SPL {X  -144.887, Y  +742.280, Z    +0.000, E1   -64.184, E3 +161458.120}
SPL {X  -140.317, Y  +751.285, Z    +0.000, E1   -63.454, E3 +161470.757}
SPL {X  -135.706, Y  +759.158, Z    +0.000, E1   -62.682, E3 +161482.158}
SPL {X  -131.040, Y  +766.207, Z    +0.000, E1   -61.854, E3 +161492.590}
SPL {X  -102.962, Y  +796.870, Z    +0.000, E1   -51.620, E3 +161617.922}
ENDSPLINE

SPLINE
SPL {X  -139.855, Y  +752.122, Z    +0.000, E1   -42.075, E3 +161740.851}
SPL {X  -153.268, Y  +720.324, Z    +0.000, E1   -30.648, E3 +161757.096}
SPL {X  -158.910, Y  +693.048, Z    +0.000, E1   -15.531, E3 +161763.167}
SPL {X  -159.977, Y  +677.095, Z    +0.000, E1    -3.968, E3 +161764.590}
SPL {X  -160.000, Y  +672.556, Z    +0.000, E1    -0.073, E3 +161764.692}
SPL {X  -160.000, Y  +669.399, Z    +0.000, E1    +3.976, E3 +161764.772}
SPL {X  -160.000, Y  +661.045, Z    +0.000, E1   +19.300, E3 +161765.361}
SPL {X  -160.000, Y  +646.999, Z    +0.000, E1   +41.048, E3 +161767.778}
SPL {X  -160.000, Y  +594.464, Z    +0.000, E1   +63.651, E3 +161788.079}
SPL {X  -160.000, Y  +465.200, Z    +0.000, E1   +67.027, E3 +161876.649}
SPL {X  -160.000, Y  +444.745, Z    +0.000, E1   +67.032, E3 +161895.058}
SPL {X  -160.000, Y  +422.224, Z    +0.000, E1   +67.044, E3 +161915.309}
ENDSPLINE

SPLINE
SPL {X  -160.000, Y  +424.635, Z    +0.000, E1   +64.425, E3 +161933.336}
ENDSPLINE

SPLINE
SPL {X  -160.000, Y  +410.501, Z    +0.000, E1   +64.162, E3 +161949.880}
SPL {X  -160.000, Y  +387.965, Z    +0.000, E1   +65.039, E3 +161965.832}
SPL {X  -158.836, Y  +366.435, Z    +0.000, E1   +65.805, E3 +161980.773}
SPL {X  -155.922, Y  +349.806, Z    +0.000, E1   +65.927, E3 +161995.420}
SPL {X  -152.875, Y  +338.486, Z    +0.000, E1   +65.488, E3 +162009.036}
SPL {X  -149.360, Y  +328.327, Z    +0.000, E1   +64.994, E3 +162021.943}
SPL {X  -145.195, Y  +318.481, Z    +0.000, E1   +64.365, E3 +162035.097}
SPL {X  -140.564, Y  +309.268, Z    +0.000, E1   +63.646, E3 +162047.917}
SPL {X  -135.770, Y  +301.044, Z    +0.000, E1   +62.840, E3 +162059.789}
SPL {X  -130.944, Y  +293.756, Z    +0.000, E1   +61.990, E3 +162070.532}
SPL {X  -103.957, Y  +264.074, Z    +0.000, E1   +52.557, E3 +162176.636}
ENDSPLINE

SPLINE
SPL {X  -133.093, Y  +296.896, Z    +0.000, E1   +44.059, E3 +162301.469}
SPL {X  -150.601, Y  +331.670, Z    +0.000, E1   +33.435, E3 +162325.732}
SPL {X  -157.739, Y  +358.898, Z    +0.000, E1   +20.026, E3 +162333.960}
SPL {X  -159.601, Y  +374.403, Z    +0.000, E1   +10.058, E3 +162336.275}
SPL {X  -159.993, Y  +384.251, Z    +0.000, E1    +2.830, E3 +162336.907}
SPL {X  -160.000, Y  +387.929, Z    +0.000, E1    -0.363, E3 +162336.976}
SPL {X  -160.000, Y  +392.137, Z    +0.000, E1    -6.580, E3 +162337.115}
SPL {X  -160.000, Y  +398.334, Z    +0.000, E1   -17.404, E3 +162337.607}
SPL {X  -160.000, Y  +410.558, Z    +0.000, E1   -36.649, E3 +162339.709}
SPL {X  -160.000, Y  +459.534, Z    +0.000, E1   -61.429, E3 +162359.304}
SPL {X  -160.000, Y  +586.246, Z    +0.000, E1   -66.315, E3 +162445.803}
SPL {X  -160.000, Y  +602.823, Z    +0.000, E1   -66.332, E3 +162461.208}
SPL {X  -160.000, Y  +621.796, Z    +0.000, E1   -66.332, E3 +162478.876}
SPL {X  -160.000, Y  +638.226, Z    +0.000, E1   -66.314, E3 +162494.204}
SPL {X  -160.000, Y  +655.092, Z    +0.000, E1   -66.336, E3 +162509.862}
SPL {X  -160.000, Y  +671.716, Z    +0.000, E1   -66.315, E3 +162525.376}
SPL {X  -159.502, Y  +687.017, Z    +0.000, E1   -66.266, E3 +162540.126}
SPL {X  -157.713, Y  +701.353, Z    +0.000, E1   -66.026, E3 +162555.353}
SPL {X  -155.081, Y  +713.767, Z    +0.000, E1   -65.665, E3 +162569.639}
SPL {X  -152.128, Y  +723.968, Z    +0.000, E1   -65.242, E3 +162582.138}
SPL {X  -148.925, Y  +732.892, Z    +0.000, E1   -64.779, E3 +162593.638}
SPL {X  -144.887, Y  +742.280, Z    +0.000, E1   -64.184, E3 +162606.268}
SPL {X  -140.317, Y  +751.285, Z    +0.000, E1   -63.454, E3 +162618.905}
SPL {X  -135.706, Y  +759.158, Z    +0.000, E1   -62.682, E3 +162630.306}
SPL {X  -131.040, Y  +766.207, Z    +0.000, E1   -61.854, E3 +162640.738}
SPL {X  -102.962, Y  +796.870, Z    +0.000, E1   -51.620, E3 +162766.070}
ENDSPLINE

SPLINE
SPL {X  -139.855, Y  +752.122, Z    +0.000, E1   -42.075, E3 +162888.998}
SPL {X  -153.268, Y  +720.324, Z    +0.000, E1   -30.648, E3 +162905.244}
SPL {X  -158.910, Y  +693.048, Z    +0.000, E1   -15.531, E3 +162911.315}
SPL {X  -159.977, Y  +677.095, Z    +0.000, E1    -3.968, E3 +162912.738}
SPL {X  -160.000, Y  +672.556, Z    +0.000, E1    -0.073, E3 +162912.840}
SPL {X  -160.000, Y  +669.399, Z    +0.000, E1    +3.976, E3 +162912.920}
SPL {X  -160.000, Y  +661.045, Z    +0.000, E1   +19.300, E3 +162913.509}
SPL {X  -160.000, Y  +646.999, Z    +0.000, E1   +41.048, E3 +162915.926}
SPL {X  -160.000, Y  +594.464, Z    +0.000, E1   +63.651, E3 +162936.227}
SPL {X  -160.000, Y  +465.200, Z    +0.000, E1   +67.027, E3 +163024.797}
SPL {X  -160.000, Y  +444.745, Z    +0.000, E1   +67.032, E3 +163043.205}
SPL {X  -160.000, Y  +422.224, Z    +0.000, E1   +67.044, E3 +163063.457}
ENDSPLINE

SPLINE
SPL {X  -160.000, Y  +424.635, Z    +0.000, E1   +64.425, E3 +163081.484}
ENDSPLINE

SPLINE
SPL {X  -160.000, Y  +410.501, Z    +0.000, E1   +64.162, E3 +163098.028}
SPL {X  -160.000, Y  +387.965, Z    +0.000, E1   +65.039, E3 +163113.980}
SPL {X  -158.836, Y  +366.435, Z    +0.000, E1   +65.805, E3 +163128.921}
SPL {X  -155.922, Y  +349.806, Z    +0.000, E1   +65.927, E3 +163143.568}
SPL {X  -152.875, Y  +338.486, Z    +0.000, E1   +65.488, E3 +163157.184}
SPL {X  -149.360, Y  +328.327, Z    +0.000, E1   +64.994, E3 +163170.091}
SPL {X  -145.195, Y  +318.481, Z    +0.000, E1   +64.365, E3 +163183.245}
SPL {X  -140.564, Y  +309.268, Z    +0.000, E1   +63.646, E3 +163196.065}
SPL {X  -135.770, Y  +301.044, Z    +0.000, E1   +62.840, E3 +163207.937}
SPL {X  -130.944, Y  +293.756, Z    +0.000, E1   +61.990, E3 +163218.680}
SPL {X  -103.957, Y  +264.074, Z    +0.000, E1   +52.557, E3 +163324.784}
ENDSPLINE

SPLINE
SPL {X  -133.093, Y  +296.896, Z    +0.000, E1   +44.059, E3 +163449.617}
SPL {X  -150.601, Y  +331.670, Z    +0.000, E1   +33.435, E3 +163473.880}
SPL {X  -157.739, Y  +358.898, Z    +0.000, E1   +20.026, E3 +163482.108}
SPL {X  -159.601, Y  +374.403, Z    +0.000, E1   +10.058, E3 +163484.423}
SPL {X  -159.993, Y  +384.251, Z    +0.000, E1    +2.830, E3 +163485.055}
SPL {X  -160.000, Y  +387.929, Z    +0.000, E1    -0.363, E3 +163485.124}
SPL {X  -160.000, Y  +392.137, Z    +0.000, E1    -6.580, E3 +163485.263}
SPL {X  -160.000, Y  +398.334, Z    +0.000, E1   -17.404, E3 +163485.754}
SPL {X  -160.000, Y  +410.558, Z    +0.000, E1   -36.649, E3 +163487.857}
SPL {X  -160.000, Y  +459.534, Z    +0.000, E1   -61.429, E3 +163507.452}
SPL {X  -160.000, Y  +586.246, Z    +0.000, E1   -66.315, E3 +163593.951}
SPL {X  -160.000, Y  +602.823, Z    +0.000, E1   -66.332, E3 +163609.355}
SPL {X  -160.000, Y  +621.796, Z    +0.000, E1   -66.332, E3 +163627.024}
SPL {X  -160.000, Y  +638.226, Z    +0.000, E1   -66.314, E3 +163642.352}
SPL {X  -160.000, Y  +655.092, Z    +0.000, E1   -66.336, E3 +163658.010}
SPL {X  -160.000, Y  +671.716, Z    +0.000, E1   -66.315, E3 +163673.524}
SPL {X  -159.502, Y  +687.017, Z    +0.000, E1   -66.266, E3 +163688.274}
SPL {X  -157.713, Y  +701.353, Z    +0.000, E1   -66.026, E3 +163703.501}
SPL {X  -155.081, Y  +713.767, Z    +0.000, E1   -65.665, E3 +163717.787}
SPL {X  -152.128, Y  +723.968, Z    +0.000, E1   -65.242, E3 +163730.286}
SPL {X  -148.925, Y  +732.892, Z    +0.000, E1   -64.779, E3 +163741.786}
SPL {X  -144.887, Y  +742.280, Z    +0.000, E1   -64.184, E3 +163754.416}
SPL {X  -140.317, Y  +751.285, Z    +0.000, E1   -63.454, E3 +163767.053}
SPL {X  -135.706, Y  +759.158, Z    +0.000, E1   -62.682, E3 +163778.454}
SPL {X  -131.040, Y  +766.207, Z    +0.000, E1   -61.854, E3 +163788.886}
SPL {X  -102.962, Y  +796.870, Z    +0.000, E1   -51.620, E3 +163914.218}
ENDSPLINE

SPLINE
SPL {X  -139.855, Y  +752.122, Z    +0.000, E1   -42.075, E3 +164037.146}
SPL {X  -153.268, Y  +720.324, Z    +0.000, E1   -30.648, E3 +164053.392}
SPL {X  -158.910, Y  +693.048, Z    +0.000, E1   -15.531, E3 +164059.463}
SPL {X  -159.977, Y  +677.095, Z    +0.000, E1    -3.968, E3 +164060.886}
SPL {X  -160.000, Y  +672.556, Z    +0.000, E1    -0.073, E3 +164060.988}
SPL {X  -160.000, Y  +669.399, Z    +0.000, E1    +3.976, E3 +164061.068}
SPL {X  -160.000, Y  +661.045, Z    +0.000, E1   +19.300, E3 +164061.657}
SPL {X  -160.000, Y  +646.999, Z    +0.000, E1   +41.048, E3 +164064.074}
SPL {X  -160.000, Y  +594.464, Z    +0.000, E1   +63.651, E3 +164084.375}
SPL {X  -160.000, Y  +465.200, Z    +0.000, E1   +67.027, E3 +164172.945}
SPL {X  -160.000, Y  +444.745, Z    +0.000, E1   +67.032, E3 +164191.353}
SPL {X  -160.000, Y  +422.224, Z    +0.000, E1   +67.044, E3 +164211.605}
ENDSPLINE

SPLINE
SPL {X  -160.000, Y  +424.635, Z    +0.000, E1   +64.425, E3 +164229.632}
ENDSPLINE

SPLINE
SPL {X  -160.000, Y  +410.501, Z    +0.000, E1   +64.162, E3 +164246.176}
SPL {X  -160.000, Y  +387.965, Z    +0.000, E1   +65.039, E3 +164262.128}
SPL {X  -158.836, Y  +366.435, Z    +0.000, E1   +65.805, E3 +164277.069}
SPL {X  -155.922, Y  +349.806, Z    +0.000, E1   +65.927, E3 +164291.715}
SPL {X  -152.875, Y  +338.486, Z    +0.000, E1   +65.488, E3 +164305.332}
SPL {X  -149.360, Y  +328.327, Z    +0.000, E1   +64.994, E3 +164318.239}
SPL {X  -145.195, Y  +318.481, Z    +0.000, E1   +64.365, E3 +164331.392}
SPL {X  -140.564, Y  +309.268, Z    +0.000, E1   +63.646, E3 +164344.213}
SPL {X  -135.770, Y  +301.044, Z    +0.000, E1   +62.840, E3 +164356.085}
SPL {X  -130.944, Y  +293.756, Z    +0.000, E1   +61.990, E3 +164366.828}
SPL {X  -103.957, Y  +264.074, Z    +0.000, E1   +52.557, E3 +164472.932}
ENDSPLINE

SPLINE
SPL {X  -133.093, Y  +296.896, Z    +0.000, E1   +44.059, E3 +164597.765}
SPL {X  -150.601, Y  +331.670, Z    +0.000, E1   +33.435, E3 +164622.028}
SPL {X  -157.739, Y  +358.898, Z    +0.000, E1   +20.026, E3 +164630.256}
SPL {X  -159.601, Y  +374.403, Z    +0.000, E1   +10.058, E3 +164632.571}
SPL {X  -159.993, Y  +384.251, Z    +0.000, E1    +2.830, E3 +164633.203}
SPL {X  -160.000, Y  +387.929, Z    +0.000, E1    -0.363, E3 +164633.272}
SPL {X  -160.000, Y  +392.137, Z    +0.000, E1    -6.580, E3 +164633.411}
SPL {X  -160.000, Y  +398.334, Z    +0.000, E1   -17.404, E3 +164633.902}
SPL {X  -160.000, Y  +410.558, Z    +0.000, E1   -36.649, E3 +164636.005}
SPL {X  -160.000, Y  +459.534, Z    +0.000, E1   -61.429, E3 +164655.600}
SPL {X  -160.000, Y  +586.246, Z    +0.000, E1   -66.315, E3 +164742.099}
SPL {X  -160.000, Y  +602.823, Z    +0.000, E1   -66.332, E3 +164757.503}
SPL {X  -160.000, Y  +621.796, Z    +0.000, E1   -66.332, E3 +164775.172}
SPL {X  -160.000, Y  +638.226, Z    +0.000, E1   -66.314, E3 +164790.500}
SPL {X  -160.000, Y  +655.092, Z    +0.000, E1   -66.336, E3 +164806.158}
SPL {X  -160.000, Y  +671.716, Z    +0.000, E1   -66.315, E3 +164821.672}
SPL {X  -159.502, Y  +687.017, Z    +0.000, E1   -66.266, E3 +164836.422}
SPL {X  -157.713, Y  +701.353, Z    +0.000, E1   -66.026, E3 +164851.649}
SPL {X  -155.081, Y  +713.767, Z    +0.000, E1   -65.665, E3 +164865.935}
SPL {X  -152.128, Y  +723.968, Z    +0.000, E1   -65.242, E3 +164878.434}
SPL {X  -148.925, Y  +732.892, Z    +0.000, E1   -64.779, E3 +164889.934}
SPL {X  -144.887, Y  +742.280, Z    +0.000, E1   -64.184, E3 +164902.564}
SPL {X  -140.317, Y  +751.285, Z    +0.000, E1   -63.454, E3 +164915.201}
SPL {X  -135.706, Y  +759.158, Z    +0.000, E1   -62.682, E3 +164926.602}
SPL {X  -131.040, Y  +766.207, Z    +0.000, E1   -61.854, E3 +164937.034}
SPL {X  -102.962, Y  +796.870, Z    +0.000, E1   -51.620, E3 +165062.366}
ENDSPLINE

SPLINE
SPL {X  -139.855, Y  +752.122, Z    +0.000, E1   -42.075, E3 +165185.294}
SPL {X  -153.268, Y  +720.324, Z    +0.000, E1   -30.648, E3 +165201.540}
SPL {X  -158.910, Y  +693.048, Z    +0.000, E1   -15.531, E3 +165207.611}
SPL {X  -159.977, Y  +677.095, Z    +0.000, E1    -3.968, E3 +165209.034}
SPL {X  -160.000, Y  +672.556, Z    +0.000, E1    -0.073, E3 +165209.136}
SPL {X  -160.000, Y  +669.399, Z    +0.000, E1    +3.976, E3 +165209.216}
SPL {X  -160.000, Y  +661.045, Z    +0.000, E1   +19.300, E3 +165209.805}
SPL {X  -160.000, Y  +646.999, Z    +0.000, E1   +41.048, E3 +165212.222}
SPL {X  -160.000, Y  +594.464, Z    +0.000, E1   +63.651, E3 +165232.523}
SPL {X  -160.000, Y  +465.200, Z    +0.000, E1   +67.027, E3 +165321.093}
SPL {X  -160.000, Y  +444.745, Z    +0.000, E1   +67.032, E3 +165339.501}
SPL {X  -160.000, Y  +422.224, Z    +0.000, E1   +67.044, E3 +165359.753}
ENDSPLINE

SPLINE
SPL {X  -160.000, Y  +424.635, Z    +0.000, E1   +64.425, E3 +165377.780}
ENDSPLINE

SPLINE
SPL {X  -160.000, Y  +410.501, Z    +0.000, E1   +64.162, E3 +165394.324}
SPL {X  -160.000, Y  +387.965, Z    +0.000, E1   +65.039, E3 +165410.276}
SPL {X  -158.836, Y  +366.435, Z    +0.000, E1   +65.805, E3 +165425.217}
SPL {X  -155.922, Y  +349.806, Z    +0.000, E1   +65.927, E3 +165439.863}
SPL {X  -152.875, Y  +338.486, Z    +0.000, E1   +65.488, E3 +165453.480}
SPL {X  -149.360, Y  +328.327, Z    +0.000, E1   +64.994, E3 +165466.387}
SPL {X  -145.195, Y  +318.481, Z    +0.000, E1   +64.365, E3 +165479.540}
SPL {X  -140.564, Y  +309.268, Z    +0.000, E1   +63.646, E3 +165492.361}
SPL {X  -135.770, Y  +301.044, Z    +0.000, E1   +62.840, E3 +165504.233}
SPL {X  -130.944, Y  +293.756, Z    +0.000, E1   +61.990, E3 +165514.976}
SPL {X  -103.957, Y  +264.074, Z    +0.000, E1   +52.557, E3 +165621.080}
ENDSPLINE

SPLINE
SPL {X  -133.093, Y  +296.896, Z    +0.000, E1   +44.059, E3 +165745.913}
SPL {X  -150.601, Y  +331.670, Z    +0.000, E1   +33.435, E3 +165770.176}
SPL {X  -157.739, Y  +358.898, Z    +0.000, E1   +20.026, E3 +165778.404}
SPL {X  -159.601, Y  +374.403, Z    +0.000, E1   +10.058, E3 +165780.719}
SPL {X  -159.993, Y  +384.251, Z    +0.000, E1    +2.830, E3 +165781.351}
SPL {X  -160.000, Y  +387.929, Z    +0.000, E1    -0.363, E3 +165781.420}
SPL {X  -160.000, Y  +392.137, Z    +0.000, E1    -6.580, E3 +165781.559}
SPL {X  -160.000, Y  +398.334, Z    +0.000, E1   -17.404, E3 +165782.050}
SPL {X  -160.000, Y  +410.558, Z    +0.000, E1   -36.649, E3 +165784.153}
SPL {X  -160.000, Y  +459.534, Z    +0.000, E1   -61.429, E3 +165803.748}
SPL {X  -160.000, Y  +586.246, Z    +0.000, E1   -66.315, E3 +165890.247}
SPL {X  -160.000, Y  +602.823, Z    +0.000, E1   -66.332, E3 +165905.651}
SPL {X  -160.000, Y  +621.796, Z    +0.000, E1   -66.332, E3 +165923.320}
SPL {X  -160.000, Y  +638.226, Z    +0.000, E1   -66.314, E3 +165938.647}
SPL {X  -160.000, Y  +655.092, Z    +0.000, E1   -66.336, E3 +165954.306}
SPL {X  -160.000, Y  +671.716, Z    +0.000, E1   -66.315, E3 +165969.820}
SPL {X  -159.502, Y  +687.017, Z    +0.000, E1   -66.266, E3 +165984.570}
SPL {X  -157.713, Y  +701.353, Z    +0.000, E1   -66.026, E3 +165999.797}
SPL {X  -155.081, Y  +713.767, Z    +0.000, E1   -65.665, E3 +166014.083}
SPL {X  -152.128, Y  +723.968, Z    +0.000, E1   -65.242, E3 +166026.582}
SPL {X  -148.925, Y  +732.892, Z    +0.000, E1   -64.779, E3 +166038.082}
SPL {X  -144.887, Y  +742.280, Z    +0.000, E1   -64.184, E3 +166050.712}
SPL {X  -140.317, Y  +751.285, Z    +0.000, E1   -63.454, E3 +166063.349}
SPL {X  -135.706, Y  +759.158, Z    +0.000, E1   -62.682, E3 +166074.750}
SPL {X  -131.040, Y  +766.207, Z    +0.000, E1   -61.854, E3 +166085.182}
SPL {X  -102.962, Y  +796.870, Z    +0.000, E1   -51.620, E3 +166210.514}
ENDSPLINE

SPLINE
SPL {X  -139.855, Y  +752.122, Z    +0.000, E1   -42.075, E3 +166333.442}
SPL {X  -153.268, Y  +720.324, Z    +0.000, E1   -30.648, E3 +166349.688}
SPL {X  -158.910, Y  +693.048, Z    +0.000, E1   -15.531, E3 +166355.759}
SPL {X  -159.977, Y  +677.095, Z    +0.000, E1    -3.968, E3 +166357.182}
SPL {X  -160.000, Y  +672.556, Z    +0.000, E1    -0.073, E3 +166357.284}
SPL {X  -160.000, Y  +669.399, Z    +0.000, E1    +3.976, E3 +166357.364}
SPL {X  -160.000, Y  +661.045, Z    +0.000, E1   +19.300, E3 +166357.953}
SPL {X  -160.000, Y  +646.999, Z    +0.000, E1   +41.048, E3 +166360.370}
SPL {X  -160.000, Y  +594.464, Z    +0.000, E1   +63.651, E3 +166380.670}
SPL {X  -160.000, Y  +465.200, Z    +0.000, E1   +67.027, E3 +166469.241}
SPL {X  -160.000, Y  +444.745, Z    +0.000, E1   +67.032, E3 +166487.649}
SPL {X  -160.000, Y  +422.224, Z    +0.000, E1   +67.044, E3 +166507.901}
ENDSPLINE

SPLINE
SPL {X  -160.000, Y  +424.635, Z    +0.000, E1   +64.425, E3 +166525.928}
ENDSPLINE

SPLINE
SPL {X  -160.000, Y  +410.501, Z    +0.000, E1   +64.162, E3 +166542.472}
SPL {X  -160.000, Y  +387.965, Z    +0.000, E1   +65.039, E3 +166558.424}
SPL {X  -158.836, Y  +366.435, Z    +0.000, E1   +65.805, E3 +166573.365}
SPL {X  -155.922, Y  +349.806, Z    +0.000, E1   +65.927, E3 +166588.011}
SPL {X  -152.875, Y  +338.486, Z    +0.000, E1   +65.488, E3 +166601.628}
SPL {X  -149.360, Y  +328.327, Z    +0.000, E1   +64.994, E3 +166614.535}
SPL {X  -145.195, Y  +318.481, Z    +0.000, E1   +64.365, E3 +166627.688}
SPL {X  -140.564, Y  +309.268, Z    +0.000, E1   +63.646, E3 +166640.509}
SPL {X  -135.770, Y  +301.044, Z    +0.000, E1   +62.840, E3 +166652.380}
SPL {X  -130.944, Y  +293.756, Z    +0.000, E1   +61.990, E3 +166663.123}
SPL {X  -103.957, Y  +264.074, Z    +0.000, E1   +52.557, E3 +166769.227}
ENDSPLINE

SPLINE
SPL {X  -133.093, Y  +296.896, Z    +0.000, E1   +44.059, E3 +166894.061}
SPL {X  -150.601, Y  +331.670, Z    +0.000, E1   +33.435, E3 +166918.324}
SPL {X  -157.739, Y  +358.898, Z    +0.000, E1   +20.026, E3 +166926.552}
SPL {X  -159.601, Y  +374.403, Z    +0.000, E1   +10.058, E3 +166928.867}
SPL {X  -159.993, Y  +384.251, Z    +0.000, E1    +2.830, E3 +166929.499}
SPL {X  -160.000, Y  +387.929, Z    +0.000, E1    -0.363, E3 +166929.568}
SPL {X  -160.000, Y  +392.137, Z    +0.000, E1    -6.580, E3 +166929.706}
SPL {X  -160.000, Y  +398.334, Z    +0.000, E1   -17.404, E3 +166930.198}
SPL {X  -160.000, Y  +410.558, Z    +0.000, E1   -36.649, E3 +166932.301}
SPL {X  -160.000, Y  +459.534, Z    +0.000, E1   -61.429, E3 +166951.896}
SPL {X  -160.000, Y  +586.246, Z    +0.000, E1   -66.315, E3 +167038.395}
SPL {X  -160.000, Y  +602.823, Z    +0.000, E1   -66.332, E3 +167053.799}
SPL {X  -160.000, Y  +621.796, Z    +0.000, E1   -66.332, E3 +167071.468}
SPL {X  -160.000, Y  +638.226, Z    +0.000, E1   -66.314, E3 +167086.795}
SPL {X  -160.000, Y  +655.092, Z    +0.000, E1   -66.336, E3 +167102.454}
SPL {X  -160.000, Y  +671.716, Z    +0.000, E1   -66.315, E3 +167117.968}
SPL {X  -159.502, Y  +687.017, Z    +0.000, E1   -66.266, E3 +167132.718}
SPL {X  -157.713, Y  +701.353, Z    +0.000, E1   -66.026, E3 +167147.945}
SPL {X  -155.081, Y  +713.767, Z    +0.000, E1   -65.665, E3 +167162.231}
SPL {X  -152.128, Y  +723.968, Z    +0.000, E1   -65.242, E3 +167174.730}
SPL {X  -148.925, Y  +732.892, Z    +0.000, E1   -64.779, E3 +167186.230}
SPL {X  -144.887, Y  +742.280, Z    +0.000, E1   -64.184, E3 +167198.860}
SPL {X  -140.317, Y  +751.285, Z    +0.000, E1   -63.454, E3 +167211.497}
SPL {X  -135.706, Y  +759.158, Z    +0.000, E1   -62.682, E3 +167222.898}
SPL {X  -131.040, Y  +766.207, Z    +0.000, E1   -61.854, E3 +167233.330}
SPL {X  -102.962, Y  +796.870, Z    +0.000, E1   -51.620, E3 +167358.662}
ENDSPLINE

SPLINE
SPL {X  -139.855, Y  +752.122, Z    +0.000, E1   -42.075, E3 +167481.590}
SPL {X  -153.268, Y  +720.324, Z    +0.000, E1   -30.648, E3 +167497.836}
SPL {X  -158.910, Y  +693.048, Z    +0.000, E1   -15.531, E3 +167503.906}
SPL {X  -159.977, Y  +677.095, Z    +0.000, E1    -3.968, E3 +167505.330}
SPL {X  -160.000, Y  +672.556, Z    +0.000, E1    -0.073, E3 +167505.432}
SPL {X  -160.000, Y  +669.399, Z    +0.000, E1    +3.976, E3 +167505.512}
SPL {X  -160.000, Y  +661.045, Z    +0.000, E1   +19.300, E3 +167506.101}
SPL {X  -160.000, Y  +646.999, Z    +0.000, E1   +41.048, E3 +167508.518}
SPL {X  -160.000, Y  +594.464, Z    +0.000, E1   +63.651, E3 +167528.818}
SPL {X  -160.000, Y  +465.200, Z    +0.000, E1   +67.027, E3 +167617.389}
SPL {X  -160.000, Y  +444.745, Z    +0.000, E1   +67.032, E3 +167635.797}
SPL {X  -160.000, Y  +422.224, Z    +0.000, E1   +67.044, E3 +167656.049}
ENDSPLINE

SPLINE
SPL {X  -160.000, Y  +424.635, Z    +0.000, E1   +64.425, E3 +167674.076}
ENDSPLINE

SPLINE
SPL {X  -160.000, Y  +410.501, Z    +0.000, E1   +64.162, E3 +167690.620}
SPL {X  -160.000, Y  +387.965, Z    +0.000, E1   +65.039, E3 +167706.572}
SPL {X  -158.836, Y  +366.435, Z    +0.000, E1   +65.805, E3 +167721.513}
SPL {X  -155.922, Y  +349.806, Z    +0.000, E1   +65.927, E3 +167736.159}
SPL {X  -152.875, Y  +338.486, Z    +0.000, E1   +65.488, E3 +167749.776}
SPL {X  -149.360, Y  +328.327, Z    +0.000, E1   +64.994, E3 +167762.683}
SPL {X  -145.195, Y  +318.481, Z    +0.000, E1   +64.365, E3 +167775.836}
SPL {X  -140.564, Y  +309.268, Z    +0.000, E1   +63.646, E3 +167788.657}
SPL {X  -135.770, Y  +301.044, Z    +0.000, E1   +62.840, E3 +167800.528}
SPL {X  -130.944, Y  +293.756, Z    +0.000, E1   +61.990, E3 +167811.271}
SPL {X  -103.957, Y  +264.074, Z    +0.000, E1   +52.557, E3 +167917.375}
ENDSPLINE

SPLINE
SPL {X  -133.093, Y  +296.896, Z    +0.000, E1   +44.059, E3 +168042.209}
SPL {X  -150.601, Y  +331.670, Z    +0.000, E1   +33.435, E3 +168066.472}
SPL {X  -157.739, Y  +358.898, Z    +0.000, E1   +20.026, E3 +168074.700}
SPL {X  -159.601, Y  +374.403, Z    +0.000, E1   +10.058, E3 +168077.015}
SPL {X  -159.993, Y  +384.251, Z    +0.000, E1    +2.830, E3 +168077.647}
SPL {X  -160.000, Y  +387.929, Z    +0.000, E1    -0.363, E3 +168077.716}
SPL {X  -160.000, Y  +392.137, Z    +0.000, E1    -6.580, E3 +168077.854}
SPL {X  -160.000, Y  +398.334, Z    +0.000, E1   -17.404, E3 +168078.346}
SPL {X  -160.000, Y  +410.558, Z    +0.000, E1   -36.649, E3 +168080.449}
SPL {X  -160.000, Y  +459.534, Z    +0.000, E1   -61.429, E3 +168100.044}
SPL {X  -160.000, Y  +586.246, Z    +0.000, E1   -66.315, E3 +168186.543}
SPL {X  -160.000, Y  +602.823, Z    +0.000, E1   -66.332, E3 +168201.947}
SPL {X  -160.000, Y  +621.796, Z    +0.000, E1   -66.332, E3 +168219.616}
SPL {X  -160.000, Y  +638.226, Z    +0.000, E1   -66.314, E3 +168234.943}
SPL {X  -160.000, Y  +655.092, Z    +0.000, E1   -66.336, E3 +168250.602}
SPL {X  -160.000, Y  +671.716, Z    +0.000, E1   -66.315, E3 +168266.116}
SPL {X  -159.502, Y  +687.017, Z    +0.000, E1   -66.266, E3 +168280.866}
SPL {X  -157.713, Y  +701.353, Z    +0.000, E1   -66.026, E3 +168296.093}
SPL {X  -155.081, Y  +713.767, Z    +0.000, E1   -65.665, E3 +168310.379}
SPL {X  -152.128, Y  +723.968, Z    +0.000, E1   -65.242, E3 +168322.878}
SPL {X  -148.925, Y  +732.892, Z    +0.000, E1   -64.779, E3 +168334.378}
SPL {X  -144.887, Y  +742.280, Z    +0.000, E1   -64.184, E3 +168347.008}
SPL {X  -140.317, Y  +751.285, Z    +0.000, E1   -63.454, E3 +168359.645}
SPL {X  -135.706, Y  +759.158, Z    +0.000, E1   -62.682, E3 +168371.046}
SPL {X  -131.040, Y  +766.207, Z    +0.000, E1   -61.854, E3 +168381.478}
SPL {X  -102.962, Y  +796.870, Z    +0.000, E1   -51.620, E3 +168506.810}
ENDSPLINE

SPLINE
SPL {X  -139.855, Y  +752.122, Z    +0.000, E1   -42.075, E3 +168629.738}
SPL {X  -153.268, Y  +720.324, Z    +0.000, E1   -30.648, E3 +168645.984}
SPL {X  -158.910, Y  +693.048, Z    +0.000, E1   -15.531, E3 +168652.054}
SPL {X  -159.977, Y  +677.095, Z    +0.000, E1    -3.968, E3 +168653.478}
SPL {X  -160.000, Y  +672.556, Z    +0.000, E1    -0.073, E3 +168653.580}
SPL {X  -160.000, Y  +669.399, Z    +0.000, E1    +3.976, E3 +168653.660}
SPL {X  -160.000, Y  +661.045, Z    +0.000, E1   +19.300, E3 +168654.249}
SPL {X  -160.000, Y  +646.999, Z    +0.000, E1   +41.048, E3 +168656.666}
SPL {X  -160.000, Y  +594.464, Z    +0.000, E1   +63.651, E3 +168676.966}
SPL {X  -160.000, Y  +465.200, Z    +0.000, E1   +67.027, E3 +168765.536}
SPL {X  -160.000, Y  +444.745, Z    +0.000, E1   +67.032, E3 +168783.945}
SPL {X  -160.000, Y  +422.224, Z    +0.000, E1   +67.044, E3 +168804.197}
ENDSPLINE

SPLINE
SPL {X  -160.000, Y  +424.635, Z    +0.000, E1   +64.425, E3 +168822.224}
ENDSPLINE

SPLINE
SPL {X  -160.000, Y  +410.501, Z    +0.000, E1   +64.162, E3 +168838.768}
SPL {X  -160.000, Y  +387.965, Z    +0.000, E1   +65.039, E3 +168854.720}
SPL {X  -158.836, Y  +366.435, Z    +0.000, E1   +65.805, E3 +168869.661}
SPL {X  -155.922, Y  +349.806, Z    +0.000, E1   +65.927, E3 +168884.307}
SPL {X  -152.875, Y  +338.486, Z    +0.000, E1   +65.488, E3 +168897.924}
SPL {X  -149.360, Y  +328.327, Z    +0.000, E1   +64.994, E3 +168910.830}
SPL {X  -145.195, Y  +318.481, Z    +0.000, E1   +64.365, E3 +168923.984}
SPL {X  -140.564, Y  +309.268, Z    +0.000, E1   +63.646, E3 +168936.805}
SPL {X  -135.770, Y  +301.044, Z    +0.000, E1   +62.840, E3 +168948.676}
SPL {X  -130.944, Y  +293.756, Z    +0.000, E1   +61.990, E3 +168959.419}
SPL {X  -103.957, Y  +264.074, Z    +0.000, E1   +52.557, E3 +169065.523}
ENDSPLINE

SPLINE
SPL {X  -133.093, Y  +296.896, Z    +0.000, E1   +44.059, E3 +169190.357}
SPL {X  -150.601, Y  +331.670, Z    +0.000, E1   +33.435, E3 +169214.620}
SPL {X  -157.739, Y  +358.898, Z    +0.000, E1   +20.026, E3 +169222.848}
SPL {X  -159.601, Y  +374.403, Z    +0.000, E1   +10.058, E3 +169225.163}
SPL {X  -159.993, Y  +384.251, Z    +0.000, E1    +2.830, E3 +169225.795}
SPL {X  -160.000, Y  +387.929, Z    +0.000, E1    -0.363, E3 +169225.864}
SPL {X  -160.000, Y  +392.137, Z    +0.000, E1    -6.580, E3 +169226.002}
SPL {X  -160.000, Y  +398.334, Z    +0.000, E1   -17.404, E3 +169226.494}
SPL {X  -160.000, Y  +410.558, Z    +0.000, E1   -36.649, E3 +169228.597}
SPL {X  -160.000, Y  +459.534, Z    +0.000, E1   -61.429, E3 +169248.192}
SPL {X  -160.000, Y  +586.246, Z    +0.000, E1   -66.315, E3 +169334.691}
SPL {X  -160.000, Y  +602.823, Z    +0.000, E1   -66.332, E3 +169350.095}
SPL {X  -160.000, Y  +621.796, Z    +0.000, E1   -66.332, E3 +169367.764}
SPL {X  -160.000, Y  +638.226, Z    +0.000, E1   -66.314, E3 +169383.091}
SPL {X  -160.000, Y  +655.092, Z    +0.000, E1   -66.336, E3 +169398.750}
SPL {X  -160.000, Y  +671.716, Z    +0.000, E1   -66.315, E3 +169414.264}
SPL {X  -159.502, Y  +687.017, Z    +0.000, E1   -66.266, E3 +169429.014}
SPL {X  -157.713, Y  +701.353, Z    +0.000, E1   -66.026, E3 +169444.241}
SPL {X  -155.081, Y  +713.767, Z    +0.000, E1   -65.665, E3 +169458.526}
SPL {X  -152.128, Y  +723.968, Z    +0.000, E1   -65.242, E3 +169471.026}
SPL {X  -148.925, Y  +732.892, Z    +0.000, E1   -64.779, E3 +169482.526}
SPL {X  -144.887, Y  +742.280, Z    +0.000, E1   -64.184, E3 +169495.156}
SPL {X  -140.317, Y  +751.285, Z    +0.000, E1   -63.454, E3 +169507.793}
SPL {X  -135.706, Y  +759.158, Z    +0.000, E1   -62.682, E3 +169519.194}
SPL {X  -131.040, Y  +766.207, Z    +0.000, E1   -61.854, E3 +169529.626}
SPL {X  -102.962, Y  +796.870, Z    +0.000, E1   -51.620, E3 +169654.958}
ENDSPLINE

SPLINE
SPL {X  -139.855, Y  +752.122, Z    +0.000, E1   -42.075, E3 +169777.886}
SPL {X  -153.268, Y  +720.324, Z    +0.000, E1   -30.648, E3 +169794.132}
SPL {X  -158.910, Y  +693.048, Z    +0.000, E1   -15.531, E3 +169800.202}
SPL {X  -159.977, Y  +677.095, Z    +0.000, E1    -3.968, E3 +169801.626}
SPL {X  -160.000, Y  +672.556, Z    +0.000, E1    -0.073, E3 +169801.728}
SPL {X  -160.000, Y  +669.399, Z    +0.000, E1    +3.976, E3 +169801.808}
SPL {X  -160.000, Y  +661.045, Z    +0.000, E1   +19.300, E3 +169802.397}
SPL {X  -160.000, Y  +646.999, Z    +0.000, E1   +41.048, E3 +169804.814}
SPL {X  -160.000, Y  +594.464, Z    +0.000, E1   +63.651, E3 +169825.114}
SPL {X  -160.000, Y  +465.200, Z    +0.000, E1   +67.027, E3 +169913.684}
SPL {X  -160.000, Y  +444.745, Z    +0.000, E1   +67.032, E3 +169932.093}
SPL {X  -160.000, Y  +422.224, Z    +0.000, E1   +67.044, E3 +169952.345}
ENDSPLINE

SPLINE
SPL {X  -160.000, Y  +424.635, Z    +0.000, E1   +64.425, E3 +169970.371}
ENDSPLINE

SPLINE
SPL {X  -160.000, Y  +410.501, Z    +0.000, E1   +64.162, E3 +169986.916}
SPL {X  -160.000, Y  +387.965, Z    +0.000, E1   +65.039, E3 +170002.868}
SPL {X  -158.836, Y  +366.435, Z    +0.000, E1   +65.805, E3 +170017.809}
SPL {X  -155.922, Y  +349.806, Z    +0.000, E1   +65.927, E3 +170032.455}
SPL {X  -152.875, Y  +338.486, Z    +0.000, E1   +65.488, E3 +170046.072}
SPL {X  -149.360, Y  +328.327, Z    +0.000, E1   +64.994, E3 +170058.978}
SPL {X  -145.195, Y  +318.481, Z    +0.000, E1   +64.365, E3 +170072.132}
SPL {X  -140.564, Y  +309.268, Z    +0.000, E1   +63.646, E3 +170084.953}
SPL {X  -135.770, Y  +301.044, Z    +0.000, E1   +62.840, E3 +170096.824}
SPL {X  -130.944, Y  +293.756, Z    +0.000, E1   +61.990, E3 +170107.567}
SPL {X  -103.957, Y  +264.074, Z    +0.000, E1   +52.557, E3 +170213.671}
ENDSPLINE

